// TIA Portal project "MOVIKIT_VELOCITY_V2.1_e_V15.1_V18" (V18)

(* hardware
DEVICE "S71500/ET200MP-Station_1"  S7-1500 station
   slot 0: "Profilschiene_0"  6ES7 590-1***0-0AA0
   slot 1: "S715xx"  CPU 1516F-3 PN/DP  6ES7 516-3FN00-0AB0  V1.8
DEVICE "SIMATIC 1200-Station_2"  S71200.Device
   slot 0: "S7-1200 Baugruppenträger"  Rack  V1.0
   slot 1: "S712xx"  CPU 1211C AC/DC/Rly  6ES7 211-1BD30-0XB0  V2.0
   slot 101: "CM 1243-5"  CM 1243-5  6GK7 243-5DX30-0XE0  V1.0
DEVICE "SIMATIC 300(1)"  S7-300 station
   slot 0: "Rack 0"  Rail  6ES7 390-1***0-0AA0
   slot 2: "CPU 315F-2 PN/DP"  CPU 315F-2 PN/DP  6ES7 315-2FH13-0AB0  V2.6
      slot 1: "MPI/DP interface_1"  X1
      slot 2: "PROFINET interface_1"  PN-IO
         slot 1: "Port_1"  Port
   slot 4: "DI 8/DO 8x24VDC/0.5A_1"  DI8/DO8 x 24VDC / 0.5A  6ES7 323-1BH01-0AA0
DEVICE "GSD-Geraet_4"  GSD.Device.PN
   slot 0: "Baugruppenträger"  Rack  V1.0
   slot 0: "velocity-s712xx"  MDX90 + CFN21 V4.0
      slot 0: "MDX90 + CFN21 V4.0"  MDX90 + CFN21 V4.0
      slot 1: "PN-IO"  PN-IO
         slot 1: "Port 1 - RJ45 (X40)"  Port 1 - RJ45 (X40)
         slot 2: "Port 2 - RJ45 (X41)"  Port 2 - RJ45 (X41)
   slot 2: "Modul I/O (05 Worte)_1"  Module I/O (05 words)
      slot 0: "Modul I/O (05 Worte)"  Module I/O (05 words)
DEVICE "GSD-Geraet_3"  GSD.Device.PN
   slot 0: "Baugruppenträger"  Rack  V1.0
   slot 0: "velocity-UDT-S715xx"  MDX90 + CFN21 V4.0
      slot 0: "MDX90 + CFN21 V4.0"  MDX90 + CFN21 V4.0
      slot 1: "PN-IO"  PN-IO
         slot 1: "Port 1 - RJ45 (X40)"  Port 1 - RJ45 (X40)
         slot 2: "Port 2 - RJ45 (X41)"  Port 2 - RJ45 (X41)
   slot 2: "Modul I/O (05 Worte)_1"  Module I/O (05 words)
      slot 0: "Modul I/O (05 Worte)"  Module I/O (05 words)
DEVICE "GSD-Geraet_2"  GSD.Device.PN
   slot 0: "Baugruppenträger"  Rack  V1.0
   slot 0: "velocity-UDT-s712xx"  MDX90 + CFN21 V4.0
      slot 0: "MDX90 + CFN21 V4.0"  MDX90 + CFN21 V4.0
      slot 1: "PN-IO"  PN-IO
         slot 1: "Port 1 - RJ45 (X40)"  Port 1 - RJ45 (X40)
         slot 2: "Port 2 - RJ45 (X41)"  Port 2 - RJ45 (X41)
   slot 2: "Modul I/O (05 Worte)_1"  Module I/O (05 words)
      slot 0: "Modul I/O (05 Worte)"  Module I/O (05 words)
   slot 3: "Modul I/O (01 Wort)_1"  Module I/O (01 word)
      slot 0: "Modul I/O (01 Wort)"  Module I/O (01 word)
   slot 4: "Modul I/O (02 Worte)_1"  Module I/O (02 words)
      slot 0: "Modul I/O (02 Worte)"  Module I/O (02 words)
   slot 5: "Modul I/O (05 Worte)_2"  Module I/O (05 words)
      slot 0: "Modul I/O (05 Worte)"  Module I/O (05 words)
DEVICE "GSD-Geraet_5"  GSD.Device.PN
   slot 0: "Baugruppenträger"  Rack  V1.0
   slot 0: "velocity-UDT-s73xx"  MDX90 + CFN21 V4.0
      slot 0: "MDX90 + CFN21 V4.0"  MDX90 + CFN21 V4.0
      slot 1: "PN-IO"  PN-IO
         slot 1: "Port 1 - RJ45 (X40)"  Port 1 - RJ45 (X40)
         slot 2: "Port 2 - RJ45 (X41)"  Port 2 - RJ45 (X41)
   slot 2: "Modul I/O (05 Worte)_1"  Module I/O (05 words)
      slot 0: "Modul I/O (05 Worte)"  Module I/O (05 words)
*)

// ===== PLC "S715xx"  CPU 1516F-3 PN/DP =====

VAR_GLOBAL   // PLC tag table "Standard-Variablentabelle"
   "Clock_Byte" AT %MB0 : Byte;
   "Clock_10Hz" AT %M0.0 : Bool;
   "Clock_5Hz" AT %M0.1 : Bool;
   "Clock_2.5Hz" AT %M0.2 : Bool;
   "Clock_2Hz" AT %M0.3 : Bool;
   "Clock_1.25Hz" AT %M0.4 : Bool;
   "Clock_1Hz" AT %M0.5 : Bool;
   "Clock_0.625Hz" AT %M0.6 : Bool;
   "Clock_0.5Hz" AT %M0.7 : Bool;
   "Reset" AT %M1000.0 : Bool;
   "set_ENABLE" AT %M1000.2 : Bool;
   "DRIVES_OFF" AT %M1000.1 : Bool;
   "VELOCITY_S715xx_Q" AT %A400.0 : "SEW_MOVIKIT_VelocityDrive_SETPOINTS_V2.1";   // Dieses UDT bildet die 5 Prozeßausgangsdaten der Funktion "Parameterkanal über Prozeßdaten" ab. This UDT maps the 5 process output data of the function "parameter channel via process data".
   "VELOCITY_S715xx_I" AT %E400.0 : "SEW_MOVIKIT_VelocityDrive_STATUS_V2.1";   // Dieses UDT bildet die 5 Prozeßeingangsdaten der Funktion "Parameterkanal über Prozeßdaten" ab. This UDT maps the 5 process input data of the function "parameter channel via process data"..
   "velocity-plus-S715xx _Start" AT %M1001.7 : Bool;
   "Status (FCB)" AT %MW1004 : Int;
   "SubFault_Fault" AT %MW1024 : Word;
   "Fault" AT %MB1024 : SInt;
   "SubFault" AT %MB1025 : SInt;
   "velocity-UDT-S715xx_PO1" AT %AW400 : Word;   // control word
   "velocity-UDT-S715xx_PO2" AT %QW402 : Int;   // setpoint speed
   "velocity-UDT-S715xx_PO3" AT %QW404 : Int;   // acceleration
   "velocity-UDT-S715xx_PO4" AT %QW406 : Int;   // deceleration
   "velocity-UDT-S715xx_PO5" AT %QW408 : Word;   // dig. Outputs
   "velocity-UDT-S715xx_PI1" AT %IW400 : Int;   // status word
   "velocity-UDT-S715xx_PI2" AT %IW402 : Int;   // actual speed
   "velocity-UDT-S715xx_PI3" AT %IW404 : Word;   // Status/Main/Subfault
   "velocity-UDT-S715xx_PI4" AT %IW406 : Int;   // actual torque
   "velocity-UDT-S715xx_PI5" AT %IW408 : Word;   // dig. Inputs
END_VAR

TYPE "SEW_MOVIKIT_VelocityDrive_STATUS_V2.1"
// Dieses UDT bildet die 5 Prozeßausgangsdaten des MOVIKIT VelocityDrives ab. This UDT maps the 5 process output data of the MOVIKIT VelocityDrive.
   STRUCT
      x_Bit_8_Fault : Bool;
      x_Bit_9_Warning : Bool;
      x_Bit_10_DriveTrain2_active : Bool;
      x_Bit_11_Setp_actual_speed_comp_signal_active : Bool;
      x_Bit_12_SW_Limit_switches_inactive : Bool;
      x_Bit_13_Reserved : Bool;
      x_Bit_14_StandBy_Mode_active : Bool;
      x_Bit_15_Heartbeat_OUT : Bool;
      x_Bit_0_Ready : Bool;
      x_Bit_1_STO_inactive : Bool;
      x_Bit_2_Output_Stage_enabled : Bool;
      x_Bit_3_Brake_released : Bool;
      x_Bit_4_Motor_turning : Bool;
      x_Bit_5_Active_Drive_referenced : Bool;
      x_Bit_6_New_Relative_Position_applied : Bool;
      x_Bit_7_In_Position : Bool;
      iActual_Speed : Int;
      wStatus_main_fault_sub_fault : Word;
      iActual_Torque : Int;
      wDigital_Inputs : Word;
   END_STRUCT;
END_TYPE

TYPE "SEW_MOVIKIT_VelocityDrive_SETPOINTS_V2.1"
TITLE = SEW_MOVIKIT_VelocityDrive_SETPOINTS
// Dieses UDT bildet die 5 Prozeßeingangsdaten des MOVIKIT VelocityDrives ab. This UDT maps the 5 process input data of the MOVIKIT VelocityDrive.
   STRUCT
      x_Bit_8_Fault_Reset : Bool;
      x_Bit_9_Reserved : Bool;
      x_Bit_10_Activate_DriveTrain2 : Bool;
      x_Bit_11_Reserved : Bool;
      x_Bit_12_Deactivate_SW_Limit_switches : Bool;
      x_Bit_13_Activate_Output_Stage_Inhibit : Bool;
      x_Bit_14_Activate_StandBy : Bool;
      x_Bit_15_Heartbeat_IN : Bool;
      x_Bit_0_Enable_Emergency_Stop : Bool;
      x_Bit_1_Enable_Application_Stop : Bool;
      x_Bit_2_Reserved : Bool;
      x_Bit_3_Release_Brake : Bool;
      x_Bit_4_Jog_positive : Bool;
      x_Bit_5_Jog_negative : Bool;
      x_Bit_6_Apply_relative_Position : Bool;
      x_Bit_7_Start_Stop : Bool;
      iSetpoint_Speed : Int;
      iAcceleration : Int;
      iDeceleration : Int;
      wDigital_Outputs : Word;
   END_STRUCT;
END_TYPE

FUNCTION "UDT_Velocity_Drive_example" : Void   // FC98, FBD
TITLE = Call the drive "velocity-UDT-S715xx"
{ S7_Optimized_Access := 'TRUE' }
AUTHOR : CSCEASDI
FAMILY : MOVIKIT
VERSION : 2.1
// This sample program only demonstrates the basic approach. We do not accept any legal or other liability for incorrect program functions and their consequences!
// 
// Please take note of the manual "MOVIKIT® Positioning, Velocity"
// 
// The UDTs "SEW_MOVIKIT_VelocityDrive_SETPOINTS_V2.1" and "SEW_MOVIKIT_VelocityDrive_STATUS_V2.1" are needed. Please make sure that the PLC data types are available in your TIA project. These UDTs can be copied from the original TIA sample project or from the MOVIKIT_VELOCITY_UDTs_V2.x.al14 library.
// 
// The plc tag "VELOCITY_S715xx_Q" has been assigned to the data type "SEW_MOVIKIT_VelocityDrive_SETPOINTS_V2.1" and  address Q400.0
// 
// The plc tag "VELOCITY_S715xx_I" has been assigned to the data type "SEW_MOVIKIT_VelocityDrive_STATUS_V2.1" and  address I400.0
BEGIN

REGION Network 1: Mapping of Status/Main fault/Subfault
   // If there is no fault or warning, the current FCB is output in "Status (FCB) MW1004 ).
   // 
   // If there is a fault or warning, the Subfault is copied in MB1024 and the Main fault in MB1025
   // 
   // => See "watch table "velocity-UDTSt15xx"
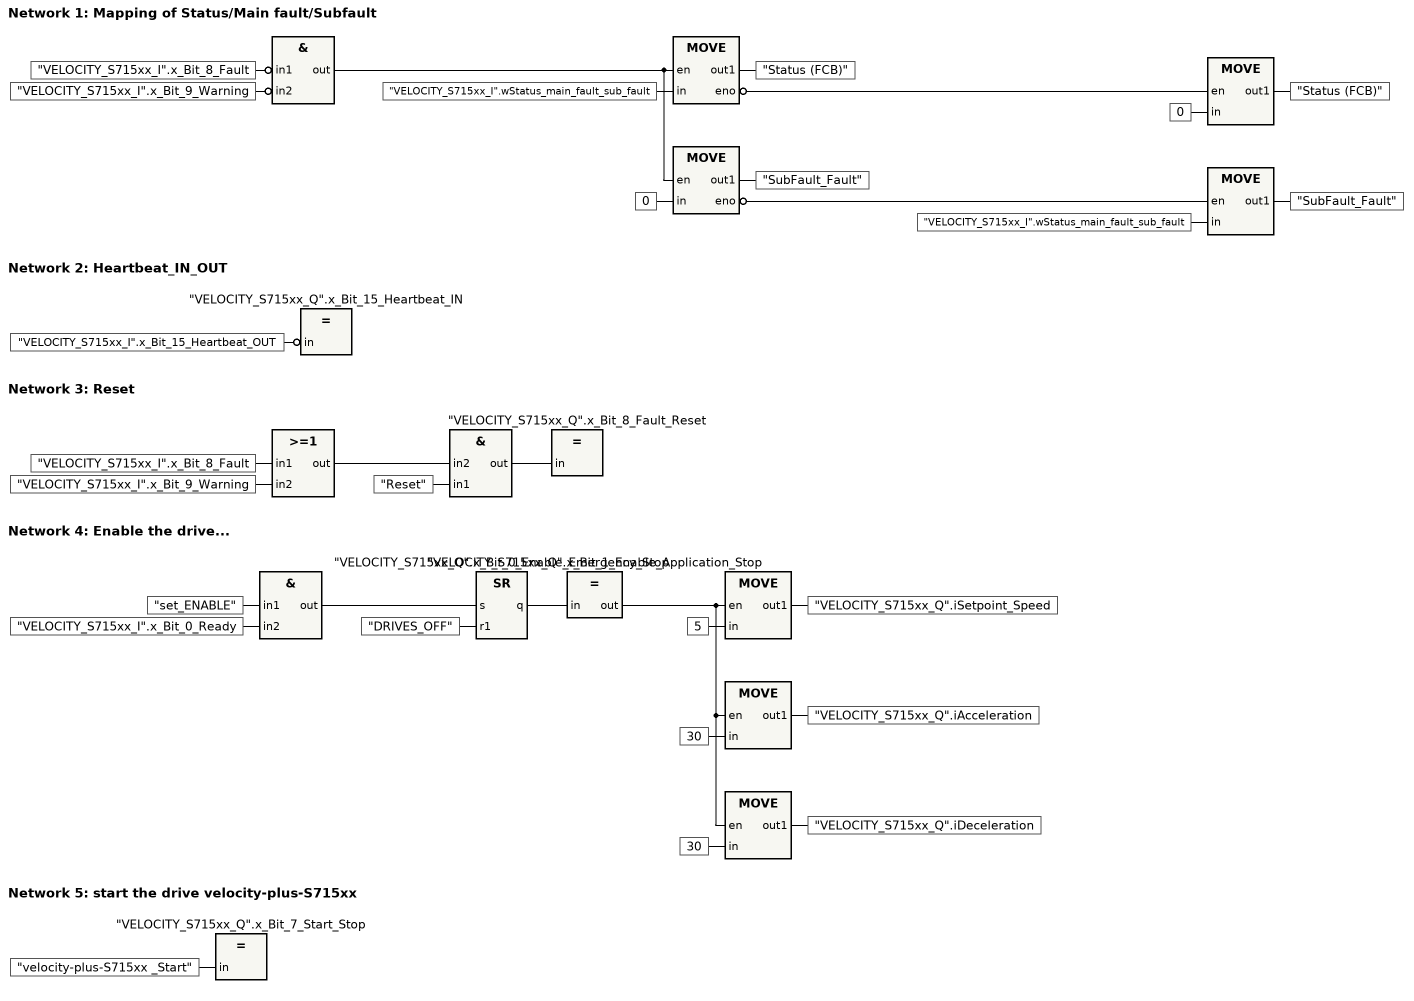
   IF NOT "VELOCITY_S715xx_I".x_Bit_8_Fault AND NOT "VELOCITY_S715xx_I".x_Bit_9_Warning THEN
       "Status (FCB)" := "VELOCITY_S715xx_I".wStatus_main_fault_sub_fault;
   END_IF;
   IF NOT (NOT "VELOCITY_S715xx_I".x_Bit_8_Fault AND NOT "VELOCITY_S715xx_I".x_Bit_9_Warning) THEN
       "Status (FCB)" := 0;
   END_IF;
   IF NOT "VELOCITY_S715xx_I".x_Bit_8_Fault AND NOT "VELOCITY_S715xx_I".x_Bit_9_Warning THEN
       "SubFault_Fault" := 0;
   END_IF;
   IF NOT (NOT "VELOCITY_S715xx_I".x_Bit_8_Fault AND NOT "VELOCITY_S715xx_I".x_Bit_9_Warning) THEN
       "SubFault_Fault" := "VELOCITY_S715xx_I".wStatus_main_fault_sub_fault;
   END_IF;
END_REGION

REGION Network 2: Heartbeat_IN_OUT
   "VELOCITY_S715xx_Q".x_Bit_15_Heartbeat_IN := NOT "VELOCITY_S715xx_I".x_Bit_15_Heartbeat_OUT;
END_REGION

REGION Network 3: Reset
   "VELOCITY_S715xx_Q".x_Bit_8_Fault_Reset := ("VELOCITY_S715xx_I".x_Bit_8_Fault OR "VELOCITY_S715xx_I".x_Bit_9_Warning) AND "Reset";
END_REGION

REGION Network 4: Enable the drive...
   // - set enable
   // - assign setpoint speed, acceleration,..,.....
   IF "set_ENABLE" AND "VELOCITY_S715xx_I".x_Bit_0_Ready THEN
       "VELOCITY_S715xx_Q".x_Bit_0_Enable_Emergency_Stop := TRUE;   // SR flip-flop
   END_IF;
   IF "DRIVES_OFF" THEN "VELOCITY_S715xx_Q".x_Bit_0_Enable_Emergency_Stop := FALSE; END_IF;
   "VELOCITY_S715xx_Q".x_Bit_1_Enable_Application_Stop := "VELOCITY_S715xx_Q".x_Bit_0_Enable_Emergency_Stop;
   IF "VELOCITY_S715xx_Q".x_Bit_0_Enable_Emergency_Stop THEN
       "VELOCITY_S715xx_Q".iSetpoint_Speed := 5;
       "VELOCITY_S715xx_Q".iAcceleration := 30;
       "VELOCITY_S715xx_Q".iDeceleration := 30;
   END_IF;
END_REGION

REGION Network 5: start the drive velocity-plus-S715xx
   "VELOCITY_S715xx_Q".x_Bit_7_Start_Stop := "velocity-plus-S715xx _Start";
END_REGION
END_FUNCTION

ORGANIZATION_BLOCK "Main"   // OB1, STL, ProgramCycle
TITLE = "Main Program Sweep (Cycle)"
{ S7_Optimized_Access := 'FALSE' }
VERSION : 0.1
// This sample program only demonstrates the basic approach. We do not accept any legal or other liability for incorrect program functions and their consequences!
// 
// Please take note of the manual "MOVIKIT® Positioning, Velocity"
   VAR_TEMP
      OB1_EV_CLASS : Byte;   // Bits 0-3 = 1 (Coming event), Bits 4-7 = 1 (Event class 1)
      OB1_SCAN_1 : Byte;   // 1 (Cold restart scan 1 of OB 1), 3 (Scan 2-n of OB 1)
      OB1_PRIORITY : Byte;   // Priority of OB Execution
      OB1_OB_NUMBR : Byte;   // 1 (Organization block 1, OB1)
      OB1_RESERVED_1 : Byte;   // Reserved for system
      OB1_RESERVED_2 : Byte;   // Reserved for system
      OB1_PREV_CYCLE : Int;   // Cycle time of previous OB1 scan (milliseconds)
      OB1_MIN_CYCLE : Int;   // Minimum cycle time of OB1 (milliseconds)
      OB1_MAX_CYCLE : Int;   // Maximum cycle time of OB1 (milliseconds)
      OB1_DATE_TIME : Date_And_Time;   // Date and time OB1 started
   END_VAR
BEGIN

REGION Network 1: Call the drive "velocity-UDT-S715xx"

         CALL  "UDT_Velocity_Drive_example";
END_REGION
END_ORGANIZATION_BLOCK

// ===== PLC "S712xx"  CPU 1211C AC/DC/Rly =====

VAR_GLOBAL   // PLC tag table "Standard-Variablentabelle"
   "Clock_Byte" AT %MB0 : Byte;
   "Clock_10Hz" AT %M0.0 : Bool;
   "Clock_5Hz" AT %M0.1 : Bool;
   "Clock_2.5Hz" AT %M0.2 : Bool;
   "Clock_2Hz" AT %M0.3 : Bool;
   "Clock_1.25Hz" AT %M0.4 : Bool;
   "Clock_1Hz" AT %M0.5 : Bool;
   "Clock_0.625Hz" AT %M0.6 : Bool;
   "Clock_0.5Hz" AT %M0.7 : Bool;
   "velocity-UDT-S712xx_PO6_Jerk_Time" AT %AW310 : Int;   // Slot 3: jerk time
   "velocity-S712xx_PO1" AT %QW326 : Int;   // control word
   "velocity-S712xx_PO2" AT %QW328 : Int;   // setpoint speed
   "velocity-S712xx_PO3" AT %QW330 : Int;   // acceleration
   "velocity-S712xx_PO4" AT %QW332 : Int;   // deceleration
   "velocity-S712xx_PO5" AT %QW334 : Int;   // dig. Outputs
   "velocity-S712xx_PI1" AT %IW326 : Int;   // status word
   "velocity-S712xx_PI2" AT %IW328 : Int;   // actual speed
   "velocity-S712xx_PI3" AT %IW330 : Int;   // Status/Main/Subfault
   "velocity-S712xx_PI4" AT %IW332 : Int;   // actual torque
   "velocity-S712xx_PI5" AT %IW334 : Int;   // dig. Inputs
   "velocity-UDT-S712xx_PO1" AT %QW300 : Int;   // Slot 2: control word
   "velocity-UDT-S712xx_PO2" AT %QW302 : Int;   // Slot 2: setpoint speed
   "velocity-UDT-S712xx_PO3" AT %QW304 : Int;   // Slot 2: acceleration
   "velocity-UDT-S712xx_PO4" AT %QW306 : Int;   // Slot 2: deceleration
   "velocity-UDT-S712xx_PO5" AT %QW308 : Int;   // Slot 2: dig. Outputs
   "velocity-UDT-S712xx_PO7" AT %QW312 : Int;   // Slot 4: control word for torque limit
   "velocity-UDT-S712xx_PO8" AT %QW314 : Int;   // Slot 4: maximum torque
   "velocity-UDT-S712xx_PO9" AT %QW316 : Int;   // Slot 5: Parameter channel control word
   "velocity-UDT-S712xx_PO10" AT %QW318 : Int;   // Slot 5: Parameter channel Index
   "velocity-UDT-S712xx_PO11" AT %QW320 : Int;   // Slot 5: Parameter channel SubIndex/Offset
   "velocity-UDT-S712xx_PO12/13" AT %QD322 : DInt;   // Slot 5: Parameter channel WriteData
   "velocity-UDT-S712xx_PI1" AT %IW300 : Int;   // Slot 2: status word
   "velocity-UDT-S712xx_PI2" AT %IW302 : Int;   // Slot 2: actual speed
   "velocity-UDT-S712xx_PI3" AT %IW304 : Int;   // Slot 2: Status/Main/Subfault
   "velocity-UDT-S712xx_PI4" AT %IW306 : Int;   // Slot 2: actual torque
   "velocity-UDT-S712xx_PI5" AT %IW308 : Int;   // Slot 2: dig. Inputs
   "velocity-UDT-S712xx_PI6" AT %IW310 : Int;   // Slot 3: res.
   "velocity-UDT-S712xx_PI7" AT %IW312 : Int;   // Slot 4: status word for torque limit
   "velocity-UDT-S712xx_PI8" AT %IW314 : Int;   // Slot 4: actual torque
   "velocity-UDT-S712xx_PI9" AT %IW316 : Int;   // Slot 5: Parameter channel status word
   "velocity-UDT-S712xx_PI10" AT %IW318 : Int;   // Slot 5: Parameter channel Index
   "velocity-UDT-S712xx_PI11" AT %IW320 : Int;   // Slot 5: Parameter channelSubIndex/Offset
   "velocity-UDT-S712xx_PI12" AT %ID322 : DInt;   // Slot 5: Parameter channel ReadData
END_VAR

TYPE "SEW_MOVIKIT_VelocityDrive_STATUS_V2.1"
// Dieses UDT bildet die 5 Prozeßausgangsdaten des MOVIKIT VelocityDrives ab. This UDT maps the 5 process output data of the MOVIKIT VelocityDrive.
   STRUCT
      x_Bit_8_Fault : Bool;
      x_Bit_9_Warning : Bool;
      x_Bit_10_DriveTrain2_active : Bool;
      x_Bit_11_Setp_actual_speed_comp_signal_active : Bool;
      x_Bit_12_SW_Limit_switches_inactive : Bool;
      x_Bit_13_Reserved : Bool;
      x_Bit_14_StandBy_Mode_active : Bool;
      x_Bit_15_Heartbeat_OUT : Bool;
      x_Bit_0_Ready : Bool;
      x_Bit_1_STO_inactive : Bool;
      x_Bit_2_Output_Stage_enabled : Bool;
      x_Bit_3_Brake_released : Bool;
      x_Bit_4_Motor_turning : Bool;
      x_Bit_5_Active_Drive_referenced : Bool;
      x_Bit_6_New_Relative_Position_applied : Bool;
      x_Bit_7_In_Position : Bool;
      iActual_Speed : Int;
      wStatus_main_fault_sub_fault : Word;
      iActual_Torque : Int;
      wDigital_Inputs : Word;
   END_STRUCT;
END_TYPE

TYPE "SEW_MOVIKIT_VelocityDrive_SETPOINTS_V2.1"
TITLE = SEW_MOVIKIT_VelocityDrive_SETPOINTS
// Dieses UDT bildet die 5 Prozeßeingangsdaten des MOVIKIT VelocityDrives ab. This UDT maps the 5 process input data of the MOVIKIT VelocityDrive.
   STRUCT
      x_Bit_8_Fault_Reset : Bool;
      x_Bit_9_Reserved : Bool;
      x_Bit_10_Activate_DriveTrain2 : Bool;
      x_Bit_11_Reserved : Bool;
      x_Bit_12_Deactivate_SW_Limit_switches : Bool;
      x_Bit_13_Activate_Output_Stage_Inhibit : Bool;
      x_Bit_14_Activate_StandBy_Mode : Bool;
      x_Bit_15_Heartbeat_IN : Bool;
      x_Bit_0_Enable_Emergency_Stop : Bool;
      x_Bit_1_Enable_Application_Stop : Bool;
      x_Bit_2_Reserved : Bool;
      x_Bit_3_Release_Brake : Bool;
      x_Bit_4_Jog_positive : Bool;
      x_Bit_5_Jog_negative : Bool;
      x_Bit_6_Apply_relative_Position : Bool;
      x_Bit_7_Start_Stop : Bool;
      iSetpoint_Speed : Int;
      iSetpoint_Acceleration : Int;
      iSetpoint_Deceleration : Int;
      wDigital_Outputs : Word;
   END_STRUCT;
END_TYPE

TYPE "SEW_MOVIKIT_5_PD_PAR_STATUS_V2.0"
   STRUCT
      x_Bit_8_READ_Service_selected : Bool;
      x_Bit_9_WRITE_Service_selected : Bool;
      x_Bit_10 : Bool;
      x_Bit_11 : Bool;
      x_Bit_12 : Bool;
      x_Bit_13_Service_active : Bool;
      x_Bit_14_Service_completed : Bool;
      x_Bit_15_Service_failed : Bool;
      x_Bit_0 : Bool;
      x_Bit_1 : Bool;
      x_Bit_2 : Bool;
      x_Bit_3 : Bool;
      x_Bit_4 : Bool;
      x_Bit_5 : Bool;
      x_Bit_6 : Bool;
      x_Bit_7 : Bool;
      i_actual_Index : Int;
      b_actual_SubIndex : Byte;
      b_actual_Offset : Byte;
      dw_value_read : DWord;
   END_STRUCT;
END_TYPE

TYPE "SEW_MOVIKIT_Function_torque_limit_STATUS_V2.0"
   STRUCT
      x_Bit_8 : Bool;
      x_Bit_9 : Bool;
      x_Bit_10 : Bool;
      x_Bit_11 : Bool;
      x_Bit_12 : Bool;
      x_Bit_13 : Bool;
      x_Bit_14 : Bool;
      x_Bit_15 : Bool;
      x_Bit_0_torque_limit_via_PD_active : Bool;
      x_Bit_1_speed_and_lag_error_monitoring_inactive : Bool;
      x_Bit_2_torque_limit_reached : Bool;
      x_Bit_3_speed_monitoring_inactive : Bool;
      x_Bit_4 : Bool;
      x_Bit_5 : Bool;
      x_Bit_6 : Bool;
      x_Bit_7 : Bool;
      i_actual_torque : Int;
   END_STRUCT;
END_TYPE

TYPE "SEW_MOVIKIT_5_PD_PAR_SETPOINTS_V2.0"
   STRUCT
      x_Bit_8_READ : Bool;
      x_Bit_9_WRITE : Bool;
      x_Bit_10 : Bool;
      x_Bit_11 : Bool;
      x_Bit_12 : Bool;
      x_Bit_13 : Bool;
      x_Bit_14_execute_function : Bool;
      x_Bit_15 : Bool;
      x_Bit_0 : Bool;
      x_Bit_1 : Bool;
      x_Bit_2 : Bool;
      x_Bit_3 : Bool;
      x_Bit_4 : Bool;
      x_Bit_5 : Bool;
      x_Bit_6 : Bool;
      x_Bit_7 : Bool;
      i_Index : Int;
      b_SubIndex : Byte;
      b_Offset : Byte;
      dw_value : DWord;
   END_STRUCT;
END_TYPE

TYPE "SEW_MOVIKIT_Function_torque_limit_SETPOINTS_V2.0"
   STRUCT
      x_Bit_8 : Bool;
      x_Bit_9 : Bool;
      x_Bit_10 : Bool;
      x_Bit_11 : Bool;
      x_Bit_12 : Bool;
      x_Bit_13 : Bool;
      x_Bit_14 : Bool;
      x_Bit_15 : Bool;
      x_Bit_0_activate_torque_limit_via_PD : Bool;
      x_Bit_1_deactivate_monitoring_of_speed_and_lag_error : Bool;
      x_Bit_2 : Bool;
      x_Bit_3_deactivate_speed_monitoring : Bool;
      x_Bit_4 : Bool;
      x_Bit_5 : Bool;
      x_Bit_6 : Bool;
      x_Bit_7 : Bool;
      i_maximum_torque : Int;
   END_STRUCT;
END_TYPE

DATA_BLOCK "Velocity_270"   // DB270
{ S7_Optimized_Access := 'FALSE' }
VERSION : 0.1
   VAR
      PO : "SEW_MOVIKIT_VelocityDrive_SETPOINTS_V2.1";
      PI : "SEW_MOVIKIT_VelocityDrive_STATUS_V2.1";
      Communication_OK : Bool;   // true: DPRD_DAT u. DPWR_DAT arbeiten fehlerfrei. false: 5-PD-Steckplatz erforderlich; Adresse an Eingang "IO_ADDRESS" überprüfen
   END_VAR
BEGIN
END_DATA_BLOCK

DATA_BLOCK "TORQUE_279"   // DB271
{ S7_Optimized_Access := 'FALSE' }
VERSION : 0.1
   VAR
      HW_IDENTIFIER : Hw_Io := 271;
      ACTIVATE_TORQUE_LIMIT_VIA_PD : Bool;
      DEACTIVATE_MONITORING_OF_SPEED_LAG_ERROR : Bool;
      DEACTIVATE_SPEED_MONITORING : Bool;
      MAXIMUM_TORQUE : Int;
      COMMUNICATION_OK : Bool;
      TORQUE_LIMIT_VIA_PD_ACTIVE : Bool;
      SPEED_LAG_ERROR_MONITORING_INACTIVE : Bool;
      TORQUE_LIMIT_REACHED : Bool;
      SPEED_MONITORING_INACTIVE : Bool;
      ACTUAL_TORQUE : Int;
   END_VAR
BEGIN
END_DATA_BLOCK

DATA_BLOCK "Velocity_290"   // DB290
{ S7_Optimized_Access := 'FALSE' }
VERSION : 0.1
   VAR
      ENABLE_RAPID_STOP : Bool;
      ENABLE_APPLICATION_STOP : Bool;
      RELEASE_BRAKE : Bool;
      START_STOP : Bool;
      RESET_ERROR : Bool;
      ACTIVATE_DRIVE_TRAIN_2 : Bool;
      DISABLE_SW_LIMIT_SWITCH : Bool;
      ACTIVATE_INHIBIT : Bool;
      ACTIVATE_STANDBY : Bool;
      SETPOINT_SPEED : Int;
      SETPOINT_ACCELERATION : Int;
      SETPOINT_DECELERATION : Int;
      DIGITAL_OUTPUTS : Word;
      COMMUNICATION_OK : Bool;
      INVERTER_READY : Bool;
      STO_INACTIVE : Bool;
      OUTPUT_STAGE_ENABLED : Bool;
      BRAKE_RELEASED : Bool;
      DRIVE_ACTIVE : Bool;
      TARGET_VALUES_ACTIVE : Bool;
      ERROR : Bool;
      WARNING : Bool;
      DRIVE_TRAIN_2_ACTIVE : Bool;
      VELOCITY_TARGET_ACTUAL_COMPARISON : Bool;
      SW_LIMIT_SWITCH_INACTIVE : Bool;
      STANDBY_ACTIVE : Bool;
      HEARTBEAT_OUT : Bool;
      ACTUAL_SPEED : Int;
      STATUS_ERROR_NO : Int;
      ACTUAL_TORQUE : Int;
      DIGITAL_INPUTS : Word;
      HEARTBEAT_IN : Bool;
   END_VAR
BEGIN
END_DATA_BLOCK

// folder: 5_PD_Parameter_channel

DATA_BLOCK "5_PD_parameter_channel_FB_DB"   // DB198
{ S7_Optimized_Access := 'FALSE' }
VERSION : 0.1
// stored: InstanceOfName 5_PD_parameter_channel_FB
"5_PD_parameter_channel_FB"
BEGIN
END_DATA_BLOCK

DATA_BLOCK "DB_5PD_PAR_272"   // DB272
{ S7_Optimized_Access := 'FALSE' }
VERSION : 0.1
   VAR
      PO : "SEW_MOVIKIT_5_PD_PAR_SETPOINTS_V2.0";
      Service : Bool;   // 0: read; 1: write
      fActivate : Bool;
      fBusy : Bool;
      fDone : Bool;
      COMMUNICATION_NOT_OK : Bool;
      TIMEOUT : Bool;
      PI : "SEW_MOVIKIT_5_PD_PAR_STATUS_V2.0";
   END_VAR
BEGIN
END_DATA_BLOCK

// folder: (top level)

FUNCTION "Call velocity-S712xx" : Void   // FC100, FBD
TITLE = Call velocity-S712xx
{ S7_Optimized_Access := 'TRUE' }
VERSION : 2.1
// This sample program only demonstrates the basic approach. We do not accept any legal or other liability for incorrect program functions and their consequences!
// 
// Please take note of the manual "MOVIKIT® Positioning, Velocity"
BEGIN

REGION Network 1: Call velocity-S712xx
   // The FC120 serves as a program module for controlling the MOVIKIT module "Velocity Drive" for the Generation C device series. With the help of the FC120, the converters can be controlled via PROFINET IO/PROFIBUS DP. 
   // 
   // Device & networks: To use this FC, a 5 PD slot must be configured.
   // 
   // Inputs of the FC:
   // 
   // "HW_Identifier": Assign the HW-Identifier of the 5 PD slot. 
   // 
   // "ENABLE_EMERGENCY_STOP" = true: Enable; false: emergency stop
   // "ENABLE_APPLICATION_STOP" = true: Enable; false: Application stop
   // "RELEASE_BRAKE" = true: release brake (without enable)
   // "START_STOP" = Start/stop with fieldbus ramp
   // "FAULT_RESET": true: Fault reset
   // "ACTIVATE_DRIVE_TRAIN_2" = true: Activate drive train 2
   // "ACTIVATE_OUPUT_STAGE_INHIBIT" = true: Activate output stage inhibit
   // "ACTIVATE_STANDBY_MODE" = true: Activate standby mode
   // "HEARTBEAT_IN": Copied to "HEARTBEAT_OUT"
   // "SETPOINT_SPEED": in user unit (INT) 
   // "SETPOINT_ACCELERATION":  in user unit (INT) 
   // "SETPOINT_DECELERATION":  in user unit (INT)
   // "DIGITAL_OUTPUTS": MoviSuite/Movikit../Inputs/Outputs: dig Outputs: the setting "control via fieldbus" is needed
   // 
   // Outputs of the FC:
   // 
   // If the data transmission/PROFINET is disrupted, all outputs will be deleted..
   // => "COMMUNICATION_OK = false (self-confirming)
   // "READY" = true: Ready for operation.
   // "STO_INACTIVE" = true: STO inactive.
   // "OUTPUT_STAGE_ENABLED" = true: Output stage enabled.
   // "BRAKE_RELEASED" = true: Brake released.
   // "MOTOR_TURNING" = true: Motor turning.
   // "FAULT" = true: Fault.
   // "WARNING" = true: Warning 
   // "DRIVE_TRAIN_2_ACTIVE" = true: Drive train 2 active.
   // "SETPOINT-ACTUAL_COMPARISON" 
   // "STANDBY_MODE_ACTIVE" = true: Stand-by Mode is active.
   // "HEARTBEAT_OUT" : This signal is copied internally from "HEARTBEAT_IN"
   // "ACTUAL_SPEED": in user unit (INT) 
   // "STATUS_MAIN_FAULT_SUB_FAULT:" (WORD)
   //    No fault: Display of current FCB; fault/warning:  High-Byte Fault; Low-Byte SubFault
   // "ACTUAL_TORQUE":in user unit (INT)
   // "DIGITAL_INPUTS" : The digital inputs are read out
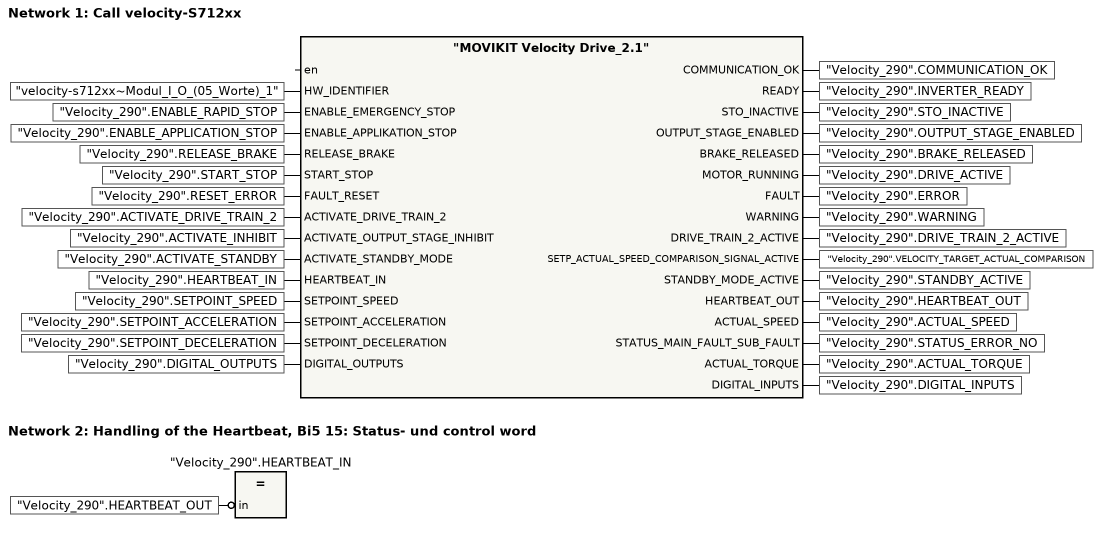
   "MOVIKIT Velocity Drive_2.1"(HW_IDENTIFIER := "velocity-s712xx~Modul_I_O_(05_Worte)_1",
                           ENABLE_EMERGENCY_STOP := "Velocity_290".ENABLE_RAPID_STOP,
                           ENABLE_APPLIKATION_STOP := "Velocity_290".ENABLE_APPLICATION_STOP,
                           RELEASE_BRAKE := "Velocity_290".RELEASE_BRAKE,
                           START_STOP := "Velocity_290".START_STOP,
                           FAULT_RESET := "Velocity_290".RESET_ERROR,
                           ACTIVATE_DRIVE_TRAIN_2 := "Velocity_290".ACTIVATE_DRIVE_TRAIN_2,
                           ACTIVATE_OUTPUT_STAGE_INHIBIT := "Velocity_290".ACTIVATE_INHIBIT,
                           ACTIVATE_STANDBY_MODE := "Velocity_290".ACTIVATE_STANDBY,
                           HEARTBEAT_IN := "Velocity_290".HEARTBEAT_IN,
                           SETPOINT_SPEED := "Velocity_290".SETPOINT_SPEED,
                           SETPOINT_ACCELERATION := "Velocity_290".SETPOINT_ACCELERATION,
                           SETPOINT_DECELERATION := "Velocity_290".SETPOINT_DECELERATION,
                           DIGITAL_OUTPUTS := "Velocity_290".DIGITAL_OUTPUTS,
                           COMMUNICATION_OK => "Velocity_290".COMMUNICATION_OK,
                           READY => "Velocity_290".INVERTER_READY,
                           STO_INACTIVE => "Velocity_290".STO_INACTIVE,
                           OUTPUT_STAGE_ENABLED => "Velocity_290".OUTPUT_STAGE_ENABLED,
                           BRAKE_RELEASED => "Velocity_290".BRAKE_RELEASED,
                           MOTOR_RUNNING => "Velocity_290".DRIVE_ACTIVE,
                           FAULT => "Velocity_290".ERROR,
                           WARNING => "Velocity_290".WARNING,
                           DRIVE_TRAIN_2_ACTIVE => "Velocity_290".DRIVE_TRAIN_2_ACTIVE,
                           SETP_ACTUAL_SPEED_COMPARISON_SIGNAL_ACTIVE => "Velocity_290".VELOCITY_TARGET_ACTUAL_COMPARISON,
                           STANDBY_MODE_ACTIVE => "Velocity_290".STANDBY_ACTIVE,
                           HEARTBEAT_OUT => "Velocity_290".HEARTBEAT_OUT,
                           ACTUAL_SPEED => "Velocity_290".ACTUAL_SPEED,
                           STATUS_MAIN_FAULT_SUB_FAULT => "Velocity_290".STATUS_ERROR_NO,
                           ACTUAL_TORQUE => "Velocity_290".ACTUAL_TORQUE,
                           DIGITAL_INPUTS => "Velocity_290".DIGITAL_INPUTS);
END_REGION

REGION Network 2: Handling of the Heartbeat, Bi5 15: Status- und control word
   "Velocity_290".HEARTBEAT_IN := NOT "Velocity_290".HEARTBEAT_OUT;
END_REGION
END_FUNCTION

FUNCTION "Call_velocity-UDT-S712xx" : Void   // FC101, FBD
TITLE = Control of the drive velocity-UDT-S712xx with the functions "Variable jerk time, Variable torque limitation.
{ S7_Optimized_Access := 'TRUE' }
VERSION : 0.1
// This sample program only demonstrates the basic approach. We do not accept any legal or other liability for incorrect program functions and their consequences!
// 
// Please take note of the manual "MOVIKIT® Positioning, Velocity"
// 
// Control of the MOVIKITS Velocity Drive with the functions "Variable jerk time and Variable torque limitation.
BEGIN

REGION Network 1: Slot 2, PD 1..5: Control of the drive velocity-UDT-S712xx
   // The FC121 serves as a program module for controlling the MOVIKIT module "Velocity Drive" for the Generation C device series. With the help of the FC121, the converters can be controlled via PROFINET IO/PROFIBUS DP. 
   // 
   // Device & networks: To use this FC, a 5 PD slot must be configured.
   // 
   // This FC uses the UDTs "SEW_MOVIKIT_VelocityDrive_SETPOINTS_V2.0" and "SEW_MOVIKIT_VelocityDrive_STATUS_V2.0". Please make sure that these PLC data types are available in your TIA project. These UDTs can be copied from the original TIA sample project or from the MOVIKIT_Vel_&_Pos_UDTs_V2.0.al14 library.
   // 
   // Inputs of the FC:
   // 
   // Attention! 
   // S71xxx: "HW_Identifier". Assign the HW-Identifier of the 5 PD slot. 
   // S73xx/4xx:"HW_Identifier"Change the data type from "HW_IO" to "WORD" Assign the peripheral address of the 5 PD slot;
   // 
   // "ENABLE_EMERGENCY_STOP" = true: Enable; false: emergency stop
   // "ENABLE_APPLICATION_STOP" = true: Enable; false: Application stop
   // "RELEASE_BRAKE" = true: release brake (without enable)
   // "START_STOP" = Start/stop with fieldbus ramp
   // "FAULT_RESET": true: Fault reset
   // "ACTIVATE_DRIVE_TRAIN_2" = true: Activate drive train 2
   // "ACTIVATE_OUPUT_STAGE_INHIBIT" = true: Activate output stage inhibit
   // "ACTIVATE_STANDBY_MODE" = true: Activate standby mode
   // "HEARTBEAT_IN": Copied to "HEARTBEAT_OUT"
   // "SETPOINT_SPEED": in user unit (INT) 
   // "SETPOINT_ACCELERATION":  in user unit (INT) 
   // "SETPOINT_DECELERATION":  in user unit (INT)
   // "DIGITAL_OUTPUTS": MoviSuite/Movikit../Inputs/Outputs: dig Outputs: the setting "control via fieldbus" is needed
   // 
   // Outputs of the FC:
   // 
   // If the data transmission/PROFINET is disrupted, all outputs will be deleted..
   // => "COMMUNICATION_OK = false (self-confirming)
   // "READY" = true: Ready for operation.
   // "STO_INACTIVE" = true: STO inactive.
   // "OUTPUT_STAGE_ENABLED" = true: Output stage enabled.
   // "BRAKE_RELEASED" = true: Brake released.
   // "MOTOR_TURNING" = true: Motor turning.
   // "FAULT" = true: Fault.
   // "WARNING" = true: Warning 
   // "DRIVE_TRAIN_2_ACTIVE" = true: Drive train 2 active.
   // "SETPOINT-ACTUAL_COMPARISON" 
   // "STANDBY_MODE_ACTIVE" = true: Stand-by Mode is active.
   // "HEARTBEAT_OUT" : This signal is copied internally from "HEARTBEAT_IN"
   // "ACTUAL_SPEED": in user unit (INT) 
   // "STATUS_MAIN_FAULT_SUB_FAULT:" (WORD)
   //    No fault: Display of current FCB; fault/warning:  High-Byte Fault; Low-Byte SubFault
   // "ACTUAL_TORQUE":in user unit (INT)
   // "DIGITAL_INPUTS" : The digital inputs are read out
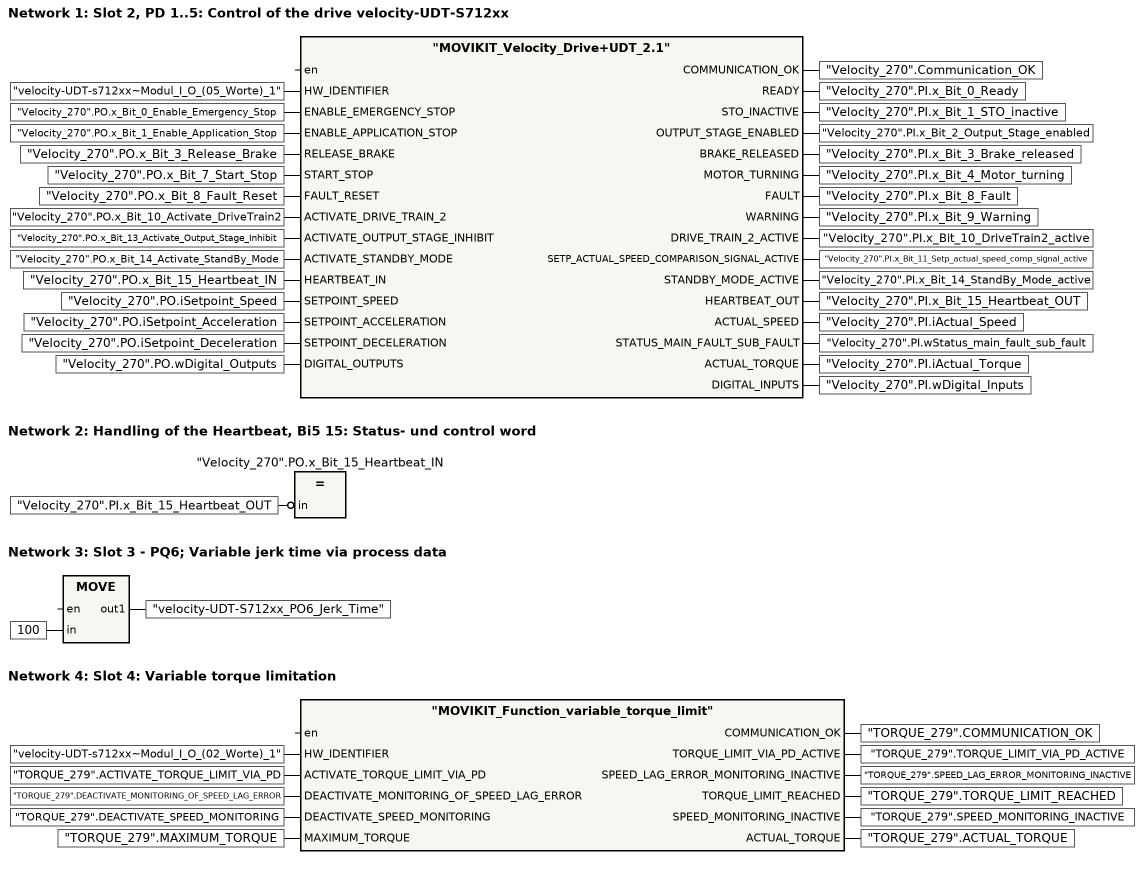
   "MOVIKIT_Velocity_Drive+UDT_2.1"(HW_IDENTIFIER := "velocity-UDT-s712xx~Modul_I_O_(05_Worte)_1",
                           ENABLE_EMERGENCY_STOP := "Velocity_270".PO.x_Bit_0_Enable_Emergency_Stop,
                           ENABLE_APPLICATION_STOP := "Velocity_270".PO.x_Bit_1_Enable_Application_Stop,
                           RELEASE_BRAKE := "Velocity_270".PO.x_Bit_3_Release_Brake,
                           START_STOP := "Velocity_270".PO.x_Bit_7_Start_Stop,
                           FAULT_RESET := "Velocity_270".PO.x_Bit_8_Fault_Reset,
                           ACTIVATE_DRIVE_TRAIN_2 := "Velocity_270".PO.x_Bit_10_Activate_DriveTrain2,
                           ACTIVATE_OUTPUT_STAGE_INHIBIT := "Velocity_270".PO.x_Bit_13_Activate_Output_Stage_Inhibit,
                           ACTIVATE_STANDBY_MODE := "Velocity_270".PO.x_Bit_14_Activate_StandBy_Mode,
                           HEARTBEAT_IN := "Velocity_270".PO.x_Bit_15_Heartbeat_IN,
                           SETPOINT_SPEED := "Velocity_270".PO.iSetpoint_Speed,
                           SETPOINT_ACCELERATION := "Velocity_270".PO.iSetpoint_Acceleration,
                           SETPOINT_DECELERATION := "Velocity_270".PO.iSetpoint_Deceleration,
                           DIGITAL_OUTPUTS := "Velocity_270".PO.wDigital_Outputs,
                           COMMUNICATION_OK => "Velocity_270".Communication_OK,
                           READY => "Velocity_270".PI.x_Bit_0_Ready,
                           STO_INACTIVE => "Velocity_270".PI.x_Bit_1_STO_inactive,
                           OUTPUT_STAGE_ENABLED => "Velocity_270".PI.x_Bit_2_Output_Stage_enabled,
                           BRAKE_RELEASED => "Velocity_270".PI.x_Bit_3_Brake_released,
                           MOTOR_TURNING => "Velocity_270".PI.x_Bit_4_Motor_turning,
                           FAULT => "Velocity_270".PI.x_Bit_8_Fault,
                           WARNING => "Velocity_270".PI.x_Bit_9_Warning,
                           DRIVE_TRAIN_2_ACTIVE => "Velocity_270".PI.x_Bit_10_DriveTrain2_active,
                           SETP_ACTUAL_SPEED_COMPARISON_SIGNAL_ACTIVE => "Velocity_270".PI.x_Bit_11_Setp_actual_speed_comp_signal_active,
                           STANDBY_MODE_ACTIVE => "Velocity_270".PI.x_Bit_14_StandBy_Mode_active,
                           HEARTBEAT_OUT => "Velocity_270".PI.x_Bit_15_Heartbeat_OUT,
                           ACTUAL_SPEED => "Velocity_270".PI.iActual_Speed,
                           STATUS_MAIN_FAULT_SUB_FAULT => "Velocity_270".PI.wStatus_main_fault_sub_fault,
                           ACTUAL_TORQUE => "Velocity_270".PI.iActual_Torque,
                           DIGITAL_INPUTS => "Velocity_270".PI.wDigital_Inputs);
END_REGION

REGION Network 2: Handling of the Heartbeat, Bi5 15: Status- und control word
   "Velocity_270".PO.x_Bit_15_Heartbeat_IN := NOT "Velocity_270".PI.x_Bit_15_Heartbeat_OUT;
END_REGION

REGION Network 3: Slot 3 - PQ6; Variable jerk time via process data
   // This additional function extends the range of functions
   // by providing the ability to specify the jerk time.
   // The additional function extends the process data
   // length by one process data word.
   // 
   // The jerk is written directly on the output word:
   "velocity-UDT-S712xx_PO6_Jerk_Time" := 100;
END_REGION

REGION Network 4: Slot 4: Variable torque limitation
   // The additional function "Variable torque limiting Q1" lets you specify the torque via the
   // application in 0.1% × nominal motor torque. For fieldbus
   // operation, the process data length is extended by 2 process data words.
   // 
   // This FC uses the UDTs "SEW_Movikit_Function_torque_limit_SETPOINTS_V2.0" and "SEW_MOVIKIT_Function_torque_limit_STATUS_V2.0". 
   // Please make sure that these PLC data types are available in your TIA project.
   // These UDTs can be copied from the original TIA sample project or from the MOVIKIT_Vel_&_Pos_UDTs_V2.0.al14 library.
   // 
   // Inputs of the FC:
   // 
   // Attention! 
   // S71xxx: "HW_Identifier". Assign the HW-Identifier of the 2 PD slot. 
   // S73xx/4xx:"HW_Identifier"Change the data type from "HW_IO" to "WORD" Assign the peripheral address of the 2 PD slot;
   // 
   // "ACTIVATE_TORQUE_LIMIT_VIA_PD": Activation of torque limiting
   // "DEACTIVATE_MONITORING_OF_SPEED_LAG_ERROR": Deactivation of monitoring for speed and lag error
   // "DEACTIVATE_SPEED_MONITORING": Deactivation of speed monitoring
   // "MAXIMUM_TORQUE": Torque related to the nominal motor torque (unit: 0.1%)
   // 
   // Outputs of the FC:
   // 
   // If the data transmission/PROFINET is disrupted, all outputs will be deleted..
   // => "COMMUNICATION_OK = false (self-confirming)
   // "TORQUE_LIMIT_VIA_PD_ACTIVE": Torque limit via PD active
   // "SPEED_LAG_ERROR_MONITORING_INACTIVE": Speed and lag error inactive
   // "TORQUE_LIMIT_REACHED": Torque limit reached
   // "SPEED_MONITORING_INACTIVE": Speed monitoring inactive
   // "ACTUAL_TORQUE": Current torque in relation to the nominal motor torque (unit: 0.1%)
   "MOVIKIT_Function_variable_torque_limit"(HW_IDENTIFIER := "velocity-UDT-s712xx~Modul_I_O_(02_Worte)_1",
                           ACTIVATE_TORQUE_LIMIT_VIA_PD := "TORQUE_279".ACTIVATE_TORQUE_LIMIT_VIA_PD,
                           DEACTIVATE_MONITORING_OF_SPEED_LAG_ERROR := "TORQUE_279".DEACTIVATE_MONITORING_OF_SPEED_LAG_ERROR,
                           DEACTIVATE_SPEED_MONITORING := "TORQUE_279".DEACTIVATE_SPEED_MONITORING,
                           MAXIMUM_TORQUE := "TORQUE_279".MAXIMUM_TORQUE,
                           COMMUNICATION_OK => "TORQUE_279".COMMUNICATION_OK,
                           TORQUE_LIMIT_VIA_PD_ACTIVE => "TORQUE_279".TORQUE_LIMIT_VIA_PD_ACTIVE,
                           SPEED_LAG_ERROR_MONITORING_INACTIVE => "TORQUE_279".SPEED_LAG_ERROR_MONITORING_INACTIVE,
                           TORQUE_LIMIT_REACHED => "TORQUE_279".TORQUE_LIMIT_REACHED,
                           SPEED_MONITORING_INACTIVE => "TORQUE_279".SPEED_MONITORING_INACTIVE,
                           ACTUAL_TORQUE => "TORQUE_279".ACTUAL_TORQUE);
END_REGION
END_FUNCTION

FUNCTION "MOVIKIT Velocity Drive_2.1" : Void   // FC120, SCL
TITLE = MOVIKIT Velocity Drive_2.1
{ S7_Optimized_Access := 'TRUE' }
AUTHOR : SVSPASE
FAMILY : MOVIKIT
VERSION : 2.1
// This sample program only demonstrates the basic approach. We do not accept any legal or other liability for incorrect program functions and their consequences!
// 
// The FC120 serves as a program module for controlling the MOVIKIT module "Velocity Drive" for the Generation C device series. With the help of the FC120,
// the converters can be controlled via PROFINET IO/PROFIBUS DP.
// 
// Device & networks: To use this FC, a 5 PD slot must be configured.
// 
// Attention Input "HW_Identifier":
// Assign the HW-Identifier of the 5 PD slot.
   VAR_INPUT
      HW_IDENTIFIER : Hw_Io;   // S71xxx: Assign the HW-Identifier of the 5 PD slot.
      ENABLE_EMERGENCY_STOP : Bool;   // true: Enable; false: emergency stop
      ENABLE_APPLIKATION_STOP : Bool;   // true: Enable; false: Application stop
      RELEASE_BRAKE : Bool;   // true: release brake (without enable)
      START_STOP : Bool;   // Start/stop with fieldbus ramp
      FAULT_RESET : Bool;   // true: Fault reset
      ACTIVATE_DRIVE_TRAIN_2 : Bool;   // true: Activate drive train 2
      ACTIVATE_OUTPUT_STAGE_INHIBIT : Bool;   // true: Activate output stage inhibit
      ACTIVATE_STANDBY_MODE : Bool;   // true: Activate standby mode
      HEARTBEAT_IN : Bool;   // Copied to HEARTBEAT_OUT
      SETPOINT_SPEED : Int;   // in user unit (INT)
      SETPOINT_ACCELERATION : Int;   // in user unit (INT)
      SETPOINT_DECELERATION : Int;   // in user unit (INT)
      DIGITAL_OUTPUTS : Word;   // MoviSuite/Movikit../Inputs/Outputs: dig Outputs: the setting "control via fieldbus" is needed
   END_VAR
   VAR_OUTPUT
      COMMUNICATION_OK : Bool;   // true: DPRD_DAT and DPWR_DAT are working correctly. false: 5 PD slot required; Check input "HW_Identifier
      READY : Bool;   // true: Ready for operation.
      STO_INACTIVE : Bool;   // true: STO inactive.
      OUTPUT_STAGE_ENABLED : Bool;   // true: Output stage enabled.
      BRAKE_RELEASED : Bool;   // true: Brake released.
      MOTOR_RUNNING : Bool;   // true: Motor running.
      FAULT : Bool;   // true: Fault.
      WARNING : Bool;   // true: Warning
      DRIVE_TRAIN_2_ACTIVE : Bool;   // true: Drive train 2 active.
      SETP_ACTUAL_SPEED_COMPARISON_SIGNAL_ACTIVE : Bool;
      STANDBY_MODE_ACTIVE : Bool;   // true: Stand-by Mode is active.
      HEARTBEAT_OUT : Bool;   // This signal is copied internally from "HEARTBEAT_IN"
      ACTUAL_SPEED : Int;   // in user unit (INT)
      STATUS_MAIN_FAULT_SUB_FAULT : Word;   // No fault: Display of current FCB; fault/warning: High-Byte Fault; Low-Byte SubFault
      ACTUAL_TORQUE : Int;   // in user unit (INT)
      DIGITAL_INPUTS : Word;   // The binary inputs are read out
   END_VAR
   VAR_TEMP
      PI : Array[1..5] of Word;
      PO : Array[1..5] of Word;
      DPRD_RET_VAL : Int;
      DPWR_RET_VAL : Int;
   END_VAR
BEGIN
   (*This sample program only demonstrates the basic approach. We do not accept any legal or other liability for incorrect program functions and their consequences!

   The FC120 serves as a program module for controlling the MOVIKIT module "Velocity Drive" for the Generation C device series. With the help of the FC120,
   the converters can be controlled via PROFINET IO/PROFIBUS DP.

   Device & networks: To use this FC, a 5 PD slot must be configured.

   Attention Input "HW_Identifier":
   Assign the HW-Identifier of the 5 PD slot. 
   *)

   //DPRD_DAT: Reading Consistent Data of a DP Standard Slave/PROFINET IO device
   #DPRD_RET_VAL:=DPRD_DAT(LADDR:=#HW_IDENTIFIER, RECORD=>#PI);


   IF #DPRD_RET_VAL = 0 THEN //If no error occurs while the instruction is being executed...

       #COMMUNICATION_OK := TRUE;

       //Mapping the signals of the Status word:
       #READY := #PI[1].%X0;
       #STO_INACTIVE := #PI[1].%X1;
       #OUTPUT_STAGE_ENABLED := #PI[1].%X2;
       #BRAKE_RELEASED := #PI[1].%X3;
       #MOTOR_RUNNING := #PI[1].%X4;
       #FAULT := #PI[1].%X8;
       #WARNING := #PI[1].%X9;
       #DRIVE_TRAIN_2_ACTIVE := #PI[1].%X10;
       #SETP_ACTUAL_SPEED_COMPARISON_SIGNAL_ACTIVE := #PI[1].%X11;
       #STANDBY_MODE_ACTIVE := #PI[1].%X14;
       #HEARTBEAT_OUT := #PI[1].%X15;

       //Assign PI2..5
       #ACTUAL_SPEED := WORD_TO_INT(#PI[2]);
       #STATUS_MAIN_FAULT_SUB_FAULT := #PI[3];
       #ACTUAL_TORQUE := WORD_TO_INT(#PI[4]) ;
       #DIGITAL_INPUTS := #PI[5];

       //Mapping the signals of the control word:
       #PO[1].%X0 := #ENABLE_EMERGENCY_STOP;
       #PO[1].%X1 := #ENABLE_APPLIKATION_STOP;
       #PO[1].%X3 := #RELEASE_BRAKE;
       #PO[1].%X7 := #START_STOP;
       #PO[1].%X8 := #FAULT_RESET;
       #PO[1].%X10 := #ACTIVATE_DRIVE_TRAIN_2;
       #PO[1].%X13 := #ACTIVATE_OUTPUT_STAGE_INHIBIT;
       #PO[1].%X14 := #ACTIVATE_STANDBY_MODE;
       #PO[1].%X15 := #HEARTBEAT_IN;

       //Set the not used Bits to "false"
       #PO[1].%X2 := FALSE;
       #PO[1].%X4 := FALSE;
       #PO[1].%X5 := FALSE;
       #PO[1].%X6 := FALSE;
       #PO[1].%X9 := FALSE;
       #PO[1].%X11 := FALSE;
       #PO[1].%X12 := FALSE;

       //Assig the POs 2..5
       #PO[2] := INT_TO_WORD(#SETPOINT_SPEED);
       #PO[3] := INT_TO_WORD(#SETPOINT_ACCELERATION);
       #PO[4] := INT_TO_WORD(#SETPOINT_DECELERATION);
       #PO[5] := #DIGITAL_OUTPUTS;

   ELSE
       GOTO END;
   END_IF;

   //DPWR_DAT: Write consistent data of a DP standard slave/PROFINET IO device
   #DPWR_RET_VAL := DPWR_DAT(LADDR := #HW_IDENTIFIER, RECORD := #PO);

   END:
   IF #DPRD_RET_VAL <> 0 OR #DPWR_RET_VAL <> 0 THEN
       #COMMUNICATION_OK := FALSE;
       //Erase FC outputs in case of an error
       #READY := FALSE;
       #STO_INACTIVE := FALSE;
       #OUTPUT_STAGE_ENABLED := FALSE;
       #BRAKE_RELEASED := FALSE;
       #MOTOR_RUNNING := FALSE;
       #FAULT := FALSE;
       #WARNING := FALSE;
       #DRIVE_TRAIN_2_ACTIVE := FALSE;
       #SETP_ACTUAL_SPEED_COMPARISON_SIGNAL_ACTIVE := FALSE;
       #STANDBY_MODE_ACTIVE := FALSE;
       #HEARTBEAT_OUT := FALSE;
       #ACTUAL_SPEED := 0;
       #STATUS_MAIN_FAULT_SUB_FAULT := 0;
       #ACTUAL_TORQUE := 0;
       #DIGITAL_INPUTS := 0;
   END_IF;
END_FUNCTION

FUNCTION "MOVIKIT_Velocity_Drive+UDT_2.1" : Void   // FC121, SCL
TITLE = Movikit_Velocity_Drive+UDT_2.1
{ S7_Optimized_Access := 'FALSE' }
AUTHOR : SVSPASE
FAMILY : MOVIKIT
VERSION : 2.1
// This sample program only demonstrates the basic approach. We do not accept any legal or other liability for incorrect program functions and their consequences!
// 
// The FC121 serves as a program module for controlling the MOVIKIT module "Velocity Drive+UDT" for the Generation C device series. With the help of the FC121,
// the converters can be controlled via PROFINET IO/PROFIBUS DP.
// 
// Device & networks: To use this FC, a 5 PD slot must be configured.
// 
// This FC uses the UDTs SEW_MOVIKIT_VelocityDrive_SETPOINTS_V2.1 and SEW_MOVIKIT_VelocityDrive_STATUS_V2.1. 
// Please make sure that these PLC data types are available in your TIA project.
// These UDTs can be copied from the original TIA sample project or from the MOVIKIT_Vel_&_Pos_UDTs_V2.x.al14 library.
// 
// Attention Input "HW_Identifier":
// Assign the HW-Identifier of the 5 PD slot. S73xx/4xx:Change Data type from HW_IO to WORD;  Assign the peripheral address of the 5 PD slot
   VAR_INPUT
      HW_IDENTIFIER : Hw_Io;   // S71xxx: Assign the HW-Identifier of the 5 PD slot. S73xx/4xx:Change Data type from HW_IO to WORD; Assign the peripheral address of the 5 PD slot
      ENABLE_EMERGENCY_STOP : Bool;   // true: Enable; false: emergency stop
      ENABLE_APPLICATION_STOP : Bool;   // true: Enable; false: Application stop
      RELEASE_BRAKE : Bool;   // true: release brake (without enable)
      START_STOP : Bool;   // Start/stop with fieldbus ramp
      FAULT_RESET : Bool;   // true: Fault reset
      ACTIVATE_DRIVE_TRAIN_2 : Bool;   // true: Activate drive train 2
      ACTIVATE_OUTPUT_STAGE_INHIBIT : Bool;   // true: Activate output stage inhibit
      ACTIVATE_STANDBY_MODE : Bool;   // true: Activate standby mode
      HEARTBEAT_IN : Bool;   // Copied to "HEARTBEAT_OUT"
      SETPOINT_SPEED : Int;   // in user unit (INT)
      SETPOINT_ACCELERATION : Int;   // in user unit (INT)
      SETPOINT_DECELERATION : Int;   // in user unit (INT)
      DIGITAL_OUTPUTS : Word;   // MoviSuite/Movikit../Inputs/Outputs: dig Outputs: the setting "control via fieldbus" is needed
   END_VAR
   VAR_OUTPUT
      COMMUNICATION_OK : Bool;   // true: DPRD_DAT and DPWR_DAT are working correctly. false: 5 PD slot required; Check input "HW_Identifier"
      READY : Bool;   // true: Ready for operation.
      STO_INACTIVE : Bool;   // true: STO inactive.
      OUTPUT_STAGE_ENABLED : Bool;   // true: Output stage enabled.
      BRAKE_RELEASED : Bool;   // true: Brake released.
      MOTOR_TURNING : Bool;   // true: Motor running.
      FAULT : Bool;   // true: Fault.
      WARNING : Bool;   // true: Warning
      DRIVE_TRAIN_2_ACTIVE : Bool;   // true: Drive train 2 active.
      SETP_ACTUAL_SPEED_COMPARISON_SIGNAL_ACTIVE : Bool;
      STANDBY_MODE_ACTIVE : Bool;   // true: Stand-by Mode is active.
      HEARTBEAT_OUT : Bool;   // This signal is copied internally from "HEARTBEAT_IN"
      ACTUAL_SPEED : Int;   // in user unit (INT)
      STATUS_MAIN_FAULT_SUB_FAULT : Word;   // No fault: Display of current FCB; fault/warning: High-Byte Fault; Low-Byte SubFault
      ACTUAL_TORQUE : Int;   // in user unit (INT)
      DIGITAL_INPUTS : Word;   // The digital inputs are read out
   END_VAR
   VAR_TEMP
      PI : "SEW_MOVIKIT_VelocityDrive_STATUS_V2.1";   // Dieses UDT bildet die 5 Prozeßeingangsdaten des MOVIKIT VelocityDrives ab. This UDT maps the 5 process input data of the MOVIKIT VelocityDrive.
      PO : "SEW_MOVIKIT_VelocityDrive_SETPOINTS_V2.1";   // Dieses UDT bildet die 5 Prozeßausgangsdaten des MOVIKIT VelocityDrives ab. This UDT maps the 5 process output data of the MOVIKIT VelocityDrive.
      DPRD_RET_VAL : Int;
      DPWR_RET_VAL : Int;
   END_VAR
BEGIN
   (*This sample program only demonstrates the basic approach. We do not accept any legal or other liability for incorrect program functions and their consequences!

   The FC121 serves as a program module for controlling the MOVIKIT module "Velocity Drive+UDT" for the Generation C device series. With the help of the FC121,
   the converters can be controlled via PROFINET IO/PROFIBUS DP.

   Device & networks: To use this FC, a 5 PD slot must be configured.

   This FC uses the UDTs SEW_MOVIKIT_VelocityDrive_SETPOINTS_V2.1 and SEW_MOVIKIT_VelocityDrive_STATUS_V2.1. 
   Please make sure that these PLC data types are available in your TIA project.
   These UDTs can be copied from the original TIA sample project or from the MOVIKIT_Vel_&_Pos_UDTs_V2.x.al14 library.

   Attention Input "HW_Identifier":
   Assign the HW-Identifier of the 5 PD slot. S73xx/4xx:Change Data type from HW_IO to WORD;  Assign the peripheral address of the 5 PD slot
   *)

   //DPRD_DAT: Reading Consistent Data of a DP Standard Slave/PROFINET IO device
   #DPRD_RET_VAL := DPRD_DAT(LADDR := #HW_IDENTIFIER, RECORD => #PI);


   IF #DPRD_RET_VAL = 0 THEN //If no error occurs while the instruction is being executed...
       #COMMUNICATION_OK := TRUE;

       //Mapping the signals of the Status word:
       #READY := #PI.x_Bit_0_Ready;
       #STO_INACTIVE := #PI.x_Bit_1_STO_inactive;
       #OUTPUT_STAGE_ENABLED := #PI.x_Bit_2_Output_Stage_enabled;
       #BRAKE_RELEASED := #PI.x_Bit_3_Brake_released;
       #MOTOR_TURNING :=#PI.x_Bit_4_Motor_turning;
       #FAULT := #PI.x_Bit_8_Fault;
       #WARNING := #PI.x_Bit_9_Warning;
       #DRIVE_TRAIN_2_ACTIVE := #PI.x_Bit_10_DriveTrain2_active;
       #SETP_ACTUAL_SPEED_COMPARISON_SIGNAL_ACTIVE := #PI.x_Bit_11_Setp_actual_speed_comp_signal_active;
       #STANDBY_MODE_ACTIVE := #PI.x_Bit_14_StandBy_Mode_active;
       #HEARTBEAT_OUT := #PI.x_Bit_15_Heartbeat_OUT;

       //Assign PI2..5
       #ACTUAL_SPEED := #PI.iActual_Speed;
       #STATUS_MAIN_FAULT_SUB_FAULT := #PI.wStatus_main_fault_sub_fault;
       #ACTUAL_TORQUE := #PI.iActual_Torque;
       #DIGITAL_INPUTS := #PI.wDigital_Inputs;

       //Mapping the signals of the control word:
       #PO.x_Bit_0_Enable_Emergency_Stop:= #ENABLE_EMERGENCY_STOP;
       #PO.x_Bit_1_Enable_Application_Stop := #ENABLE_APPLICATION_STOP;
       #PO.x_Bit_3_Release_Brake:= #RELEASE_BRAKE;
       #PO.x_Bit_7_Start_Stop:= #START_STOP;
       #PO.x_Bit_8_Fault_Reset := #FAULT_RESET;
       #PO.x_Bit_10_Activate_DriveTrain2 := #ACTIVATE_DRIVE_TRAIN_2;
       #PO.x_Bit_13_Activate_Output_Stage_Inhibit := #ACTIVATE_OUTPUT_STAGE_INHIBIT;
       #PO.x_Bit_14_Activate_StandBy_Mode := #ACTIVATE_STANDBY_MODE;
       #PO.x_Bit_15_Heartbeat_IN := #HEARTBEAT_IN;

       //Set the not used Bits to "false"
       #PO.x_Bit_2_Reserved:= FALSE;
       #PO.x_Bit_4_Jog_positive := FALSE;
       #PO.x_Bit_5_Jog_negative  := FALSE;
       #PO.x_Bit_6_Apply_relative_Position := FALSE;
       #PO.x_Bit_9_Reserved := FALSE;
       #PO.x_Bit_11_Reserved := FALSE;
       #PO.x_Bit_12_Deactivate_SW_Limit_switches := false;

       //Assig the POs 2..5
       #PO.iSetpoint_Speed := #SETPOINT_SPEED;
       #PO.iSetpoint_Acceleration := #SETPOINT_ACCELERATION;
       #PO.iSetpoint_Deceleration := #SETPOINT_DECELERATION;
       #PO.wDigital_Outputs := #DIGITAL_OUTPUTS;

   ELSE
       GOTO END;
   END_IF;

   //DPWR_DAT: Write consistent data of a DP standard slave/PROFINET IO device
   #DPWR_RET_VAL := DPWR_DAT(LADDR := #HW_IDENTIFIER, RECORD := #PO);

   END:
   IF #DPRD_RET_VAL <> 0 OR #DPWR_RET_VAL <> 0 THEN
       #COMMUNICATION_OK := FALSE;
       //Erase FC outputs in case of an error
       #READY := FALSE;
       #STO_INACTIVE := FALSE;
       #OUTPUT_STAGE_ENABLED := FALSE;
       #BRAKE_RELEASED := FALSE;
       #MOTOR_TURNING := FALSE;
       #FAULT := FALSE;
       #WARNING := FALSE;
       #DRIVE_TRAIN_2_ACTIVE := FALSE;
       #SETP_ACTUAL_SPEED_COMPARISON_SIGNAL_ACTIVE := FALSE;
       #STANDBY_MODE_ACTIVE := FALSE;
       #HEARTBEAT_OUT := FALSE;
       #ACTUAL_SPEED := 0;
       #STATUS_MAIN_FAULT_SUB_FAULT := 0;
       #ACTUAL_TORQUE := 0;
       #DIGITAL_INPUTS := 0;
   END_IF;
END_FUNCTION

FUNCTION "MOVIKIT_Function_variable_torque_limit" : Void   // FC191, SCL
TITLE = Movikit_Function_variable_torque_limit
{ S7_Optimized_Access := 'FALSE' }
AUTHOR : SVSPASE
FAMILY : MOVIKIT
VERSION : 2.0
// This sample program only demonstrates the basic approach. We do not accept any legal or other liability for incorrect program functions and their consequences!
// 
// This FC is used to control the MOVIKIT function "variable torque limit Q1 (2PD)"
// 
// Device & networks: To use this FC, a 2 PD slot must be configured.
// 
// This FC uses the UDTs "SEW_Movikit_Function_torque_limit_SETPOINTS_V2.0" and "SEW_MOVIKIT_Function_torque_limit_STATUS_V2.0". 
// Please make sure that these PLC data types are available in your TIA project.
// These UDTs can be copied from the original TIA sample project or from the MOVIKIT_Vel_&_Pos_UDTs_V2.0.al14 library.
// 
// Attention Input "HW_Identifier":
// Assign the HW-Identifier of the 2 PD slot. S73xx/4xx:Change Data type from HW_IO to WORD;  Assign the peripheral address of the 2 PD slot
   VAR_INPUT
      HW_IDENTIFIER : Hw_Io;   // S71xxx: Assign the HW-Identifier of the 2 PD slot. S73xx/4xx:Change Data type from HW_IO to WORD; Assign the peripheral address of the 2 PD slot
      ACTIVATE_TORQUE_LIMIT_VIA_PD : Bool;   // activate torque limit via PD
      DEACTIVATE_MONITORING_OF_SPEED_LAG_ERROR : Bool;   // deactivate monitoring of lag and speed errors
      DEACTIVATE_SPEED_MONITORING : Bool;   // deactivate speed monitoring
      MAXIMUM_TORQUE : Int;   // maximum torque
   END_VAR
   VAR_OUTPUT
      COMMUNICATION_OK : Bool;
      TORQUE_LIMIT_VIA_PD_ACTIVE : Bool;   // Torque limit via PD active
      SPEED_LAG_ERROR_MONITORING_INACTIVE : Bool;   // Speed and lag error inactive
      TORQUE_LIMIT_REACHED : Bool;   // Torque limit reached
      SPEED_MONITORING_INACTIVE : Bool;   // Speed monitoring inactive
      ACTUAL_TORQUE : Int;   // Actual torque
   END_VAR
   VAR_TEMP
      PI : "SEW_MOVIKIT_Function_torque_limit_STATUS_V2.0";
      PO : "SEW_MOVIKIT_Function_torque_limit_SETPOINTS_V2.0";
      DPRD_RET_VAL : Int;
      DPWR_RET_VAL : Int;
   END_VAR
BEGIN
   (*This sample program only demonstrates the basic approach. We do not accept any legal or other liability for incorrect program functions and their consequences!

   This FC is used to control the MOVIKIT function "variable torque limit Q1 (2PD)"

   Device & networks: To use this FC, a 2 PD slot must be configured.

   This FC uses the UDTs "SEW_Movikit_Function_torque_limit_SETPOINTS_V2.0" and "SEW_MOVIKIT_Function_torque_limit_STATUS_V2.0". 
   Please make sure that these PLC data types are available in your TIA project.
   These UDTs can be copied from the original TIA sample project or from the MOVIKIT_Vel_&_Pos_UDTs_V2.0.al14 library.

   Attention Input "HW_Identifier":
   Assign the HW-Identifier of the 2 PD slot. S73xx/4xx:Change Data type from HW_IO to WORD;  Assign the peripheral address of the 2 PD slot*)



   //DPWR_DAT: Write consistent data of a DP standard slave/PROFINET IO device
   #DPRD_RET_VAL := DPRD_DAT(LADDR := #HW_IDENTIFIER, RECORD => #PI);


   IF #DPRD_RET_VAL = 0 THEN
       #COMMUNICATION_OK := TRUE;

       //Mapping the signals of the Status word:
       #TORQUE_LIMIT_VIA_PD_ACTIVE := #PI.x_Bit_0_torque_limit_via_PD_active;
       #SPEED_LAG_ERROR_MONITORING_INACTIVE := #PI.x_Bit_1_speed_and_lag_error_monitoring_inactive;
       #TORQUE_LIMIT_REACHED := #PI.x_Bit_2_torque_limit_reached;
       #SPEED_MONITORING_INACTIVE := #PI.x_Bit_3_speed_monitoring_inactive;

       //Zuweisen der Ausgangsworte des Bausteins
       #ACTUAL_TORQUE := #PI.i_actual_torque;

       //Mapping the signals of the control word:
       #PO.x_Bit_0_activate_torque_limit_via_PD := #ACTIVATE_TORQUE_LIMIT_VIA_PD;
       #PO.x_Bit_1_deactivate_monitoring_of_speed_and_lag_error:= #DEACTIVATE_MONITORING_OF_SPEED_LAG_ERROR;
       #PO.x_Bit_3_deactivate_speed_monitoring := #DEACTIVATE_SPEED_MONITORING;

       //Set the not used Bits to "false"
       #PO.x_Bit_2 := FALSE;
       #PO.x_Bit_4:= FALSE;
       #PO.x_Bit_5:= FALSE;
       #PO.x_Bit_6 := FALSE;
       #PO.x_Bit_7 := FALSE;
       #PO.x_Bit_8 := FALSE;
       #PO.x_Bit_9 := FALSE;
       #PO.x_Bit_10:= FALSE;
       #PO.x_Bit_11:= FALSE;
       #PO.x_Bit_12:= FALSE;
       #PO.x_Bit_13:= FALSE;
       #PO.x_Bit_14:= FALSE;
       #PO.x_Bit_15:= FALSE;

       #PO.i_maximum_torque := #MAXIMUM_TORQUE;

   ELSE
       GOTO END;
   END_IF;

   //DPWR_DAT: Write consistent data of a DP standard slave/PROFINET IO device
   #DPWR_RET_VAL := DPWR_DAT(LADDR := #HW_IDENTIFIER, RECORD := #PO);

   END:
   IF #DPRD_RET_VAL <> 0 OR #DPWR_RET_VAL <> 0 THEN
       #COMMUNICATION_OK := FALSE;

       //Erase FC outputs in case of an error
       #TORQUE_LIMIT_VIA_PD_ACTIVE := FALSE;
       #SPEED_LAG_ERROR_MONITORING_INACTIVE := FALSE;
       #TORQUE_LIMIT_REACHED := FALSE;
       #SPEED_MONITORING_INACTIVE := FALSE;

       #ACTUAL_TORQUE := 0;
   END_IF;
END_FUNCTION

ORGANIZATION_BLOCK "Main"   // OB1, FBD, ProgramCycle
TITLE = "Main Program Sweep (Cycle)"
{ S7_Optimized_Access := 'TRUE' }
VERSION : 0.1
// This sample program only demonstrates the basic approach. We do not accept any legal or other liability for incorrect program functions and their consequences!
// 
// Please take note of the manual "MOVIKIT® Positioning, Velocity"
BEGIN

REGION Network 1: Control of the drive velocity-UDT-S712xx with the functions "Variable jerk time, Variable torque limitation, parameter channel via process data (5PD).
   // Control of the drive velocity-UDT-S712xx with the functions "Variable jerk time, Variable torque limitation, parameter channel via process data (5PD).
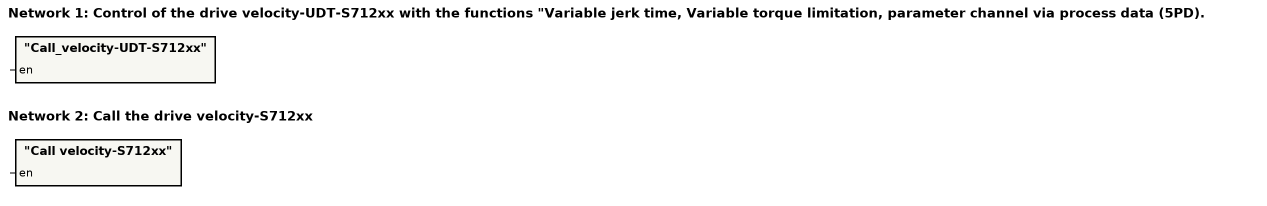
   "Call_velocity-UDT-S712xx"();
END_REGION

REGION Network 2: Call the drive velocity-S712xx
   // without the use of UDTs, without the functions "Variable jerk time, Variable torque limitation, parameter channel via process data (5PD)
   "Call velocity-S712xx"();
END_REGION
END_ORGANIZATION_BLOCK

// folder: 5_PD_Parameter_channel

FUNCTION_BLOCK "5_PD_parameter_channel_FB"   // FB198, SCL
TITLE = 5_PD_parameter_channel_FB
{ S7_Optimized_Access := 'FALSE' }
AUTHOR : SVSPASE
FAMILY : MOVIKIT
VERSION : 2.0
// This sample program only demonstrates the basic approach. We do not accept any legal or other liability for incorrect program functions and their consequences!
// 
// This FB is used to control the MOVIKIT function "parameter channel via process dada (5PD)"
// 
// Device & networks: To use this FB, a 5 PD slot must be configured.
// 
// This FC uses the UDTs "SEW_MOVIKIT_5_PD_PAR_SETPOINTS_V2.0" and "SEW_MOVIKIT_5_PD_PAR_STATUS_V2.0". 
// Please make sure that these PLC data types are available in your TIA project. 
// These UDTs can be copied from the original TIA sample project or from the MOVIKIT_Vel_&_Pos_UDTs_V2.0.al14 library.
// 
// Attention Input "HW_Identifier":
// Assign the HW-Identifier of the 5 PD slot. S73xx/4xx:Change Data type from HW_IO to WORD;  Assign the peripheral address of the 5 PD slot
   VAR_INPUT
      HW_Identifier : Hw_Io;   // S71xxx: Assign the HW-Identifier of the 5 PD slot. S73xx/4xx:Change Data type from HW_IO to WORD; Assign the peripheral address of the 5 PD slot
      SERVICE : Bool;   // false: READ; true: WRITE
      INDEX : Int;   // Index
      SubIndex : Byte;   // Subindex
      OFFSET : Byte;   // Offset
      WRITE_DATA : DWord;   // value to write
   END_VAR
   VAR_OUTPUT
      COMMUNICATION_NOT_OK : Bool;   // true: DPRD_DAT and DPWR_DAT are not working correctly. 5 PD slot required; Check input "HW_Identifier"
      TIMEOUT : Bool;   // true: the participant does not respond.
      READ_SERVICE_SELECTED : Bool;   // "Read" service selected
      WRITE_SERVICE_SELECTED : Bool;   // "Write" service selected
      ERROR : Bool;   // Service failed
      ACTUAL_INDEX : Int;   // selected Index
      ACTUAL_SUBINDEX : Byte;   // selected Subindex
      ACTUAL_OFFSET : Byte;   // selected Offset
      READ_DATA_OR_ERROR_CODE : DWord;   // Read value or error code at Error = true; Error codes are documented in the manual "MOVIKIT POSITIONING VELOCITY DRIVE"
   END_VAR
   VAR_IN_OUT
      ACTIVATE : Bool;   // activate a parameter service
      BUSY : Bool;   // the parameter service is busy right now
      DONE : Bool;   // a parameter service is done
   END_VAR
   VAR
      PI : "SEW_MOVIKIT_5_PD_PAR_STATUS_V2.0";
      PO : "SEW_MOVIKIT_5_PD_PAR_SETPOINTS_V2.0";
      DPRD_RET_VAL : Int;
      DPWR_RET_VAL : Int;
      TimeoutCounter : Int := 1000;
   END_VAR
BEGIN
   (*This sample program only demonstrates the basic approach. We do not accept any legal or other liability for incorrect program functions and their consequences!

   This FB198 serves as a program block for controlling the MOVIKIT function "Parameter channel via process data 5PD)" for the generation C device series,
   Which is implemented up to Movi-C main firmware 9.00.
   Device & networks: To use this FB, a 5 PD slot must be configured.

   This FC uses the UDTs "SEW_MOVIKIT_5_PD_PAR_SETPOINTS_V2.0" and "SEW_MOVIKIT_5_PD_PAR_STATUS_V2.0". 
   Please make sure that these PLC data types are available in your TIA project. 
   These UDTs can be copied from the original TIA sample project or from the MOVIKIT_Vel_&_Pos_UDTs_V2.0.al14 library.

   Attention Input "HW_Identifier":
   Assign the HW-Identifier of the 5 PD slot. S73xx/4xx:Change Data type from HW_IO to WORD;  Assign the peripheral address of the 5 PD slot*)


   IF #ACTIVATE THEN //Initilization
       #ACTIVATE := false; 
       #BUSY := true;
       #DONE := false;
       #TIMEOUT := false;
       #TimeoutCounter := 1000;

   //Assign the POs:
       IF #SERVICE = false THEN //Read service
           #PO.x_Bit_8_READ := true;
           #PO.x_Bit_9_WRITE := false;
       ELSE
           #PO.x_Bit_8_READ:= false;
           #PO.x_Bit_9_WRITE :=true; //Write service
       END_IF;

       #PO.x_Bit_14_execute_function:= false; //Prepare positive signal edge
       #PO.i_Index := #INDEX;
       #PO.b_Offset := #OFFSET;
       #PO.b_SubIndex:= #SubIndex;
       #PO.dw_value:=#WRITE_DATA;

     //Write the init. values: DPWR_DAT: Write consistent data of a DP standard slave/PROFINET IO device
       #DPWR_RET_VAL := DPWR_DAT(LADDR := #HW_Identifier, RECORD := #PO);
      RETURN; // //exit the FB; end of the init. 
   END_IF;


   IF #BUSY = 1 THEN
       //Timeout monitoring
       #TimeoutCounter := #TimeoutCounter - 1;
       IF #TimeoutCounter = 0 THEN
           #ERROR := true;
           #BUSY := false;
           #DONE := true;
           #TIMEOUT := true;
           #READ_DATA_OR_ERROR_CODE := 0;
           RETURN; //exit the FB
       END_IF;


           #DPRD_RET_VAL := DPRD_DAT(LADDR := #HW_Identifier, RECORD => #PI);   //DPRD_DAT: Read consistent data of a DP standard slave
           IF #DPRD_RET_VAL = 0 THEN
               #COMMUNICATION_NOT_OK := 0; 

               IF #INDEX = #PI.i_actual_Index THEN                 //Check whether the parameter channel already reports back the sent data           
                   #PO.x_Bit_14_execute_function := true;  

                   IF #PI.x_Bit_14_Service_completed = true THEN  //If "Service is completed" the parameter service is "done"..
                               #BUSY := false;
                               #DONE := true;

                   END_IF;
     //Mapping of the process input data   
                   #READ_SERVICE_SELECTED := #PI.x_Bit_8_READ_Service_selected;
                   #WRITE_SERVICE_SELECTED := #PI.x_Bit_9_WRITE_Service_selected;
                   #ERROR := #PI.x_Bit_15_Service_failed;
                   #ACTUAL_INDEX := #PI.i_actual_Index;
                   #ACTUAL_OFFSET := #PI.b_actual_Offset; //WORD_TO_INT(#PI[3] AND w#16#ff);//Hide the high-byte
                   #ACTUAL_SUBINDEX := #PI.b_actual_SubIndex;//WORD_TO_INT(SHR(IN := #PI[3], N := 8)); //shift 8 Bits/1 Byte right...
                   #READ_DATA_OR_ERROR_CODE := #PI.dw_value_read;
       END_IF;

       #DPWR_RET_VAL := DPWR_DAT(LADDR := #HW_Identifier, RECORD := #PO); //DPWR_DAT: Write consistent data of a DP standard slave/PROFINET IO device

       ELSE
           GOTO END;
       END_IF; 

       END:
       IF #DPRD_RET_VAL <> 0 OR #DPWR_RET_VAL <> 0  THEN
               #BUSY := false;
               #DONE := true;
               #ERROR := true;
               #COMMUNICATION_NOT_OK := 1;
               //Erase FB outputs in case of an error
               #READ_SERVICE_SELECTED := false;
               #WRITE_SERVICE_SELECTED := false;
               #ACTUAL_INDEX := 0;
               #ACTUAL_SUBINDEX := 0;
               #ACTUAL_OFFSET := 0;
               #READ_DATA_OR_ERROR_CODE := 0;
           END_IF;
       END_IF;  //Busy
END_FUNCTION_BLOCK

FUNCTION "Call velocity-UDT-S712xx_parameter channel via process data (5PD)" : Void   // FC105, FBD
TITLE = Call 5 PD Parameter channel
{ S7_Optimized_Access := 'TRUE' }
VERSION : 0.1
// This sample program only demonstrates the basic approach. We do not accept any legal or other liability for incorrect program functions and their consequences!
// 
// This FB198 serves as a program block for controlling the MOVIKIT function "Parameter channel via process data 5PD)" for the generation C device series,
// which is implemented up to Movi-C main firmware 9.00.
// Device & networks: To use this FB, a 5 PD slot must be configured.
BEGIN

REGION Network 1: Slot 5; Reading the head sink temperature - Mapping of Index & SubIndex
   // MoviSuite: Diagnostics/Process values/Output stage/Utilization/Heat sink temperature; 
   // Index 8312; SubIndex 5
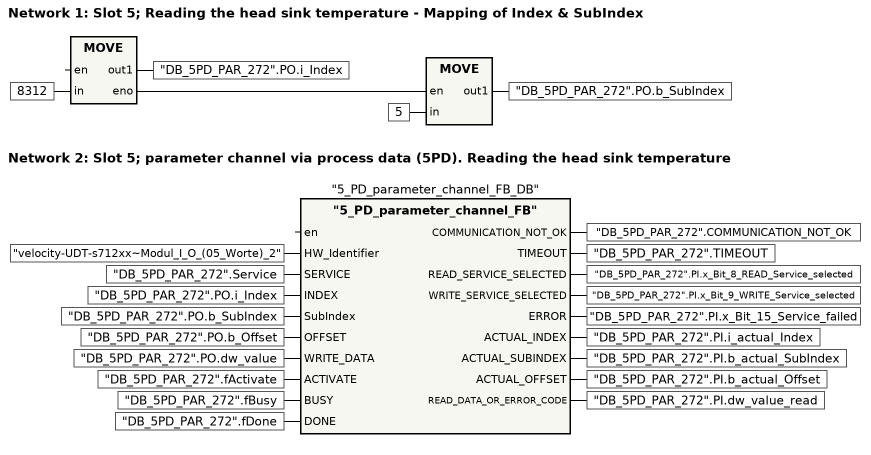
   // ENO of a box is taken as its EN; it also drops when the box reports an error
   "DB_5PD_PAR_272".PO.i_Index := 8312;
   "DB_5PD_PAR_272".PO.b_SubIndex := 5;
END_REGION

REGION Network 2: Slot 5; parameter channel via process data (5PD). Reading the head sink temperature
   // MoviSuite: Diagnostics/Process values/Output stage/Utilization/Heat sink temperature; 
   // Index 8312; SubIndex 5 
   // 
   // With this additional function, parameters can be read and written volatile.
   // The Additional function extends the process data length by 5 process data words.
   // 
   // Inputs of the FB:
   // 
   // Attention! 
   // S71xxx: "HW_Identifier". Assign the HW-Identifier of the 5 PD slot. 
   // S73xx/4xx:"HW_Identifier"Change the data type from "HW_IO" to "WORD" Assign the peripheral address of the 5 PD slot;
   // 
   // "SERVICE": false: READ; true: WRITE
   // "INDEX": Index
   // "SubIndex": Subindex
   // "OFFSET": Offset
   // "WRITE_DATA": value to write
   // 
   // 
   // Outputs of the FB:
   // 
   // "COMMUNICATION_NOT_OK": true: DPRD_DAT and DPWR_DAT are not working correctly. 5 PD slot required; 
   //                                                    Check input  "HW_Identifier"
   // "TIMEOUT": true: true:  the participant does not respond.
   // "READ_SERVICE_SELECTED": "Read" service selected
   // "WRITE_SERVICE_SELECTED": "Write" service selected
   // "ERROR": Service failed
   // "ACTUAL_INDEX": selected Index
   // "ACTUAL_SUBINDEX": selected Subindex
   // "ACTUAL_OFFSET": selected Offset
   // "READ_DATA_OR_ERROR_CODE": Read value or error code at Error = true; Error codes are documented in the manual                                                           "MOVIKIT POSITIONING VELOCITY DRIVE"
   // 
   // Status machine of the FB:
   // ACTIVATE: activate a parameter service
   // BUSY: the parameter service is busy right now
   // DONE: a parameter service is done
   "5_PD_parameter_channel_FB_DB"(HW_Identifier := "velocity-UDT-s712xx~Modul_I_O_(05_Worte)_2",   // "5_PD_parameter_channel_FB"
                           SERVICE := "DB_5PD_PAR_272".Service,
                           INDEX := "DB_5PD_PAR_272".PO.i_Index,
                           SubIndex := "DB_5PD_PAR_272".PO.b_SubIndex,
                           OFFSET := "DB_5PD_PAR_272".PO.b_Offset,
                           WRITE_DATA := "DB_5PD_PAR_272".PO.dw_value,
                           ACTIVATE := "DB_5PD_PAR_272".fActivate,
                           BUSY := "DB_5PD_PAR_272".fBusy,
                           DONE := "DB_5PD_PAR_272".fDone,
                           COMMUNICATION_NOT_OK => "DB_5PD_PAR_272".COMMUNICATION_NOT_OK,
                           TIMEOUT => "DB_5PD_PAR_272".TIMEOUT,
                           READ_SERVICE_SELECTED => "DB_5PD_PAR_272".PI.x_Bit_8_READ_Service_selected,
                           WRITE_SERVICE_SELECTED => "DB_5PD_PAR_272".PI.x_Bit_9_WRITE_Service_selected,
                           ERROR => "DB_5PD_PAR_272".PI.x_Bit_15_Service_failed,
                           ACTUAL_INDEX => "DB_5PD_PAR_272".PI.i_actual_Index,
                           ACTUAL_SUBINDEX => "DB_5PD_PAR_272".PI.b_actual_SubIndex,
                           ACTUAL_OFFSET => "DB_5PD_PAR_272".PI.b_actual_Offset,
                           READ_DATA_OR_ERROR_CODE => "DB_5PD_PAR_272".PI.dw_value_read);
END_REGION
END_FUNCTION

// ===== PLC "CPU 315F-2 PN/DP"  CPU 315F-2 PN/DP =====

VAR_GLOBAL   // PLC tag table "Standard-Variablentabelle"
   "Clock_0.5Hz" AT %M0.7 : Bool;
   "Clock_Byte" AT %MB0 : Byte;
   "Clock_10Hz" AT %M0.0 : Bool;
   "Clock_5Hz" AT %M0.1 : Bool;
   "Clock_2.5Hz" AT %M0.2 : Bool;
   "Clock_2Hz" AT %M0.3 : Bool;
   "Clock_1.25Hz" AT %M0.4 : Bool;
   "Clock_1Hz" AT %M0.5 : Bool;
   "Clock_0.625Hz" AT %M0.6 : Bool;
   "velocity-UDT-S73xx_PO1" AT %AW300 : Word;   // control word
   "velocity-UDT-S73xx_PO2" AT %QW302 : Word;   // setpoint speed
   "velocity-UDT-S73xx_PO3" AT %QW304 : Word;   // acceleration
   "velocity-UDT-S73xx_PO4" AT %QW306 : Word;   // deceleration
   "velocity-UDT-S73xx_PO5" AT %QW308 : Word;   // dig. Outputs
   "velocity-UDT-S73xx_PI1" AT %IW300 : Word;   // status word
   "velocity-UDT-S73xx_PI2" AT %IW302 : Word;   // actual speed
   "velocity-UDT-S73xx_PI3" AT %IW304 : Word;   // Status/Main/Subfault
   "velocity-UDT-S73xx_PI4" AT %IW306 : Word;   // actual torque
   "velocity-UDT-S73xx_PI5" AT %IW308 : Word;   // dig. Inputs
END_VAR

TYPE "SEW_MOVIKIT_VelocityDrive_STATUS_V2.1"
// Dieses UDT bildet die 5 Prozeßausgangsdaten des MOVIKIT VelocityDrives ab. This UDT maps the 5 process output data of the MOVIKIT VelocityDrive.
   STRUCT
      x_Bit_8_Fault : Bool;
      x_Bit_9_Warning : Bool;
      x_Bit_10_DriveTrain2_active : Bool;
      x_Bit_11_Setp_actual_speed_comp_signal_active : Bool;
      x_Bit_12_SW_Limit_switches_inactive : Bool;
      x_Bit_13_Reserved : Bool;
      x_Bit_14_StandBy_Mode_active : Bool;
      x_Bit_15_Heartbeat_OUT : Bool;
      x_Bit_0_Ready : Bool;
      x_Bit_1_STO_inactive : Bool;
      x_Bit_2_Output_Stage_enabled : Bool;
      x_Bit_3_Brake_released : Bool;
      x_Bit_4_Motor_turning : Bool;
      x_Bit_5_Active_Drive_referenced : Bool;
      x_Bit_6_New_Relative_Position_applied : Bool;
      x_Bit_7_In_Position : Bool;
      iActual_Speed : Int;
      wStatus_main_fault_sub_fault : Word;
      iActual_Torque : Int;
      wDigital_Inputs : Word;
   END_STRUCT;
END_TYPE

TYPE "SEW_MOVIKIT_VelocityDrive_SETPOINTS_V2.1"
TITLE = SEW_MOVIKIT_VelocityDrive_SETPOINTS
// Dieses UDT bildet die 5 Prozeßeingangsdaten des MOVIKIT VelocityDrives ab. This UDT maps the 5 process input data of the MOVIKIT VelocityDrive.
   STRUCT
      x_Bit_8_Fault_Reset : Bool;
      x_Bit_9_Reserved : Bool;
      x_Bit_10_Activate_DriveTrain2 : Bool;
      x_Bit_11_Reserved : Bool;
      x_Bit_12_Deactivate_SW_Limit_switches : Bool;
      x_Bit_13_Activate_Output_Stage_Inhibit : Bool;
      x_Bit_14_Activate_StandBy : Bool;
      x_Bit_15_Heartbeat_IN : Bool;
      x_Bit_0_Enable_Emergency_Stop : Bool;
      x_Bit_1_Enable_Application_Stop : Bool;
      x_Bit_2_Reserved : Bool;
      x_Bit_3_Release_Brake : Bool;
      x_Bit_4_Jog_positive : Bool;
      x_Bit_5_Jog_negative : Bool;
      x_Bit_6_Apply_relative_Position : Bool;
      x_Bit_7_Start_Stop : Bool;
      iSetpoint_Speed : Int;
      iAcceleration : Int;
      iDeceleration : Int;
      wDigital_Outputs : Word;
   END_STRUCT;
END_TYPE

DATA_BLOCK "MOVIKIT_Velocity_256"   // DB256
{ S7_Optimized_Access := 'FALSE' }
VERSION : 0.1
   VAR
      PO : "SEW_MOVIKIT_VelocityDrive_SETPOINTS_V2.1";
      PI : "SEW_MOVIKIT_VelocityDrive_STATUS_V2.1";
      Communication_OK : Bool;   // true: DPRD_DAT and DPWR_DAT are working correctly. false: 5 PD slot required; Check address at Input "IO_ADDRESS"
   END_VAR
BEGIN
END_DATA_BLOCK

FUNCTION "Call_Velocity_UDT_S73xx" : Void   // FC100, FBD
TITLE = Call_Velocity_UDT_S73xx
{ S7_Optimized_Access := 'FALSE' }
VERSION : 0.1
// This sample program only demonstrates the basic approach. We do not accept any legal or other liability for incorrect program functions and their consequences!
// 
// Please take note of the manual "MOVIKIT® Positioning, Velocity"
BEGIN

REGION Network 1: Control of the drive velocity-UDT-S73xx
   // The FC122 serves as a program module for controlling the MOVIKIT module "Velocity Drive" for the Generation C device series. With the help of the FC122, the converters can be controlled via PROFINET IO/PROFIBUS DP. 
   // 
   // Device & networks: To use this FC, a 5 PD slot must be configured.
   // 
   // This FC uses the UDTs "SEW_MOVIKIT_VelocityDrive_SETPOINTS_V2.1" and "SEW_MOVIKIT_VelocityDrive_STATUS_V2.1". Please make sure that these PLC data types are available in your TIA project. These UDTs can be copied from the original TIA sample project or from the MOVIKIT_Vel_&_Pos_UDTs_V2.x.al14 library.
   // 
   // Inputs of the FC:
   // 
   // Attention! 
   // S73xx/4xx:"IO_ADDRESS"/Data Type Word:  Assign the peripheral address of the 5 PD slot;
   // S71xxx: "IO_ADDRESS" change the data type from Word to "HW_IO". Assign the HW-Identifier of the 5 PD slot. 
   // 
   // "ENABLE_EMERGENCY_STOP" = true: Enable; false: emergency stop
   // "ENABLE_APPLICATION_STOP" = true: Enable; false: Application stop
   // "RELEASE_BRAKE" = true: release brake (without enable)
   // "START_STOP" = Start/stop with fieldbus ramp
   // "FAULT_RESET": true: Fault reset
   // "ACTIVATE_DRIVE_TRAIN_2" = true: Activate drive train 2
   // "ACTIVATE_OUPUT_STAGE_INHIBIT" = true: Activate output stage inhibit
   // "ACTIVATE_STANDBY_MODE" = true: Activate standby mode
   // "HEARTBEAT_IN": Copied to "HEARTBEAT_OUT"
   // "SETPOINT_SPEED": in user unit (INT) 
   // "SETPOINT_ACCELERATION":  in user unit (INT) 
   // "SETPOINT_DECELERATION":  in user unit (INT)
   // "DIGITAL_OUTPUTS": MoviSuite/Movikit../Inputs/Outputs: dig Outputs: the setting "control via fieldbus" is needed
   // 
   // Outputs of the FC:
   // 
   // If the data transmission/PROFINET is disrupted, all outputs will be deleted..
   // => "COMMUNICATION_OK = false (self-confirming)
   // "READY" = true: Ready for operation.
   // "STO_INACTIVE" = true: STO inactive.
   // "OUTPUT_STAGE_ENABLED" = true: Output stage enabled.
   // "BRAKE_RELEASED" = true: Brake released.
   // "MOTOR_TURNING" = true: Motor turning.
   // "FAULT" = true: Fault.
   // "WARNING" = true: Warning 
   // "DRIVE_TRAIN_2_ACTIVE" = true: Drive train 2 active.
   // "SETPOINT-ACTUAL_COMPARISON" 
   // "STANDBY_MODE_ACTIVE" = true: Stand-by Mode is active.
   // "HEARTBEAT_OUT" : This signal is copied internally from "HEARTBEAT_IN"
   // "ACTUAL_SPEED": in user unit (INT) 
   // "STATUS_MAIN_FAULT_SUB_FAULT:" (WORD)
   //    No fault: Display of current FCB; fault/warning:  High-Byte Fault; Low-Byte SubFault
   // "ACTUAL_TORQUE":in user unit (INT)
   // "DIGITAL_INPUTS" : The digital inputs are read out
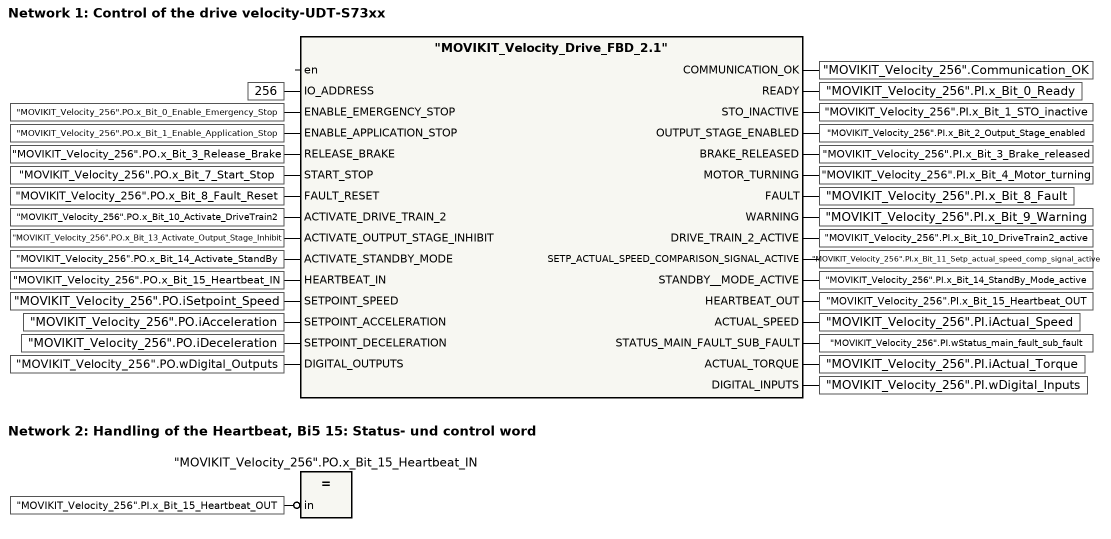
   "MOVIKIT_Velocity_Drive_FBD_2.1"(IO_ADDRESS := 256,
                           ENABLE_EMERGENCY_STOP := "MOVIKIT_Velocity_256".PO.x_Bit_0_Enable_Emergency_Stop,
                           ENABLE_APPLICATION_STOP := "MOVIKIT_Velocity_256".PO.x_Bit_1_Enable_Application_Stop,
                           RELEASE_BRAKE := "MOVIKIT_Velocity_256".PO.x_Bit_3_Release_Brake,
                           START_STOP := "MOVIKIT_Velocity_256".PO.x_Bit_7_Start_Stop,
                           FAULT_RESET := "MOVIKIT_Velocity_256".PO.x_Bit_8_Fault_Reset,
                           ACTIVATE_DRIVE_TRAIN_2 := "MOVIKIT_Velocity_256".PO.x_Bit_10_Activate_DriveTrain2,
                           ACTIVATE_OUTPUT_STAGE_INHIBIT := "MOVIKIT_Velocity_256".PO.x_Bit_13_Activate_Output_Stage_Inhibit,
                           ACTIVATE_STANDBY_MODE := "MOVIKIT_Velocity_256".PO.x_Bit_14_Activate_StandBy,
                           HEARTBEAT_IN := "MOVIKIT_Velocity_256".PO.x_Bit_15_Heartbeat_IN,
                           SETPOINT_SPEED := "MOVIKIT_Velocity_256".PO.iSetpoint_Speed,
                           SETPOINT_ACCELERATION := "MOVIKIT_Velocity_256".PO.iAcceleration,
                           SETPOINT_DECELERATION := "MOVIKIT_Velocity_256".PO.iDeceleration,
                           DIGITAL_OUTPUTS := "MOVIKIT_Velocity_256".PO.wDigital_Outputs,
                           COMMUNICATION_OK => "MOVIKIT_Velocity_256".Communication_OK,
                           READY => "MOVIKIT_Velocity_256".PI.x_Bit_0_Ready,
                           STO_INACTIVE => "MOVIKIT_Velocity_256".PI.x_Bit_1_STO_inactive,
                           OUTPUT_STAGE_ENABLED => "MOVIKIT_Velocity_256".PI.x_Bit_2_Output_Stage_enabled,
                           BRAKE_RELEASED => "MOVIKIT_Velocity_256".PI.x_Bit_3_Brake_released,
                           MOTOR_TURNING => "MOVIKIT_Velocity_256".PI.x_Bit_4_Motor_turning,
                           FAULT => "MOVIKIT_Velocity_256".PI.x_Bit_8_Fault,
                           WARNING => "MOVIKIT_Velocity_256".PI.x_Bit_9_Warning,
                           DRIVE_TRAIN_2_ACTIVE => "MOVIKIT_Velocity_256".PI.x_Bit_10_DriveTrain2_active,
                           SETP_ACTUAL_SPEED_COMPARISON_SIGNAL_ACTIVE => "MOVIKIT_Velocity_256".PI.x_Bit_11_Setp_actual_speed_comp_signal_active,
                           STANDBY__MODE_ACTIVE => "MOVIKIT_Velocity_256".PI.x_Bit_14_StandBy_Mode_active,
                           HEARTBEAT_OUT => "MOVIKIT_Velocity_256".PI.x_Bit_15_Heartbeat_OUT,
                           ACTUAL_SPEED => "MOVIKIT_Velocity_256".PI.iActual_Speed,
                           STATUS_MAIN_FAULT_SUB_FAULT => "MOVIKIT_Velocity_256".PI.wStatus_main_fault_sub_fault,
                           ACTUAL_TORQUE => "MOVIKIT_Velocity_256".PI.iActual_Torque,
                           DIGITAL_INPUTS => "MOVIKIT_Velocity_256".PI.wDigital_Inputs);
END_REGION

REGION Network 2: Handling of the Heartbeat, Bi5 15: Status- und control word
   "MOVIKIT_Velocity_256".PO.x_Bit_15_Heartbeat_IN := NOT "MOVIKIT_Velocity_256".PI.x_Bit_15_Heartbeat_OUT;
END_REGION
END_FUNCTION

FUNCTION "MOVIKIT_Velocity_Drive_FBD_2.1" : Void   // FC122, FBD
TITLE = MOVIKIT Velocity Drive/S73xx in FBD_2.1
{ S7_Optimized_Access := 'FALSE' }
AUTHOR : CSCEASDI
FAMILY : MOVIKIT
VERSION : 2.1
// This sample program only demonstrates the basic approach. We do not accept any legal or other liability for incorrect program functions and their consequences!
// 
// The FC122 serves as a program module for controlling the MOVIKIT module "Velocity Drive" for the Generation C device series. With the help of the FC122, the converters can be controlled via PROFINET IO/PROFIBUS DP. 
// 
// Device & networks: To use this FC, a 5 PD slot must be configured.
// 
// This FC uses the UDTs SEW_MOVIKIT_VelocityDrive_SETPOINTS_V2.0 and SEW_MOVIKIT_VelocityDrive_STATUS_V2.0. Please make sure that these PLC data types are available in your TIA project. These UDTs can be copied from the original TIA sample project or from the MOVIKIT_Vel_&_Pos_UDTs_V2.0.al14 library.
// 
// Attention! 
// S73xx/4xx:"IO_ADDRESS"/Data Type Word:  Assign the peripheral address of the 5 PD slot;
// S71xxx: "IO_ADDRESS" change the data type from Word to "HW_IO". Assign the HW-Identifier of the 5 PD slot.
   VAR_INPUT
      IO_ADDRESS : Word;   // S73xx/4xx:"IO_ADDRESS"/Data Type Word: Assign the peripheral address of the 5 PD slot; S71xxx: "IO_ADDRESS" change the data type from Word to "HW_IO". Assign the HW-Identifier of the 5 PD slot.
      ENABLE_EMERGENCY_STOP : Bool;   // true: Enable; false: emergency stop
      ENABLE_APPLICATION_STOP : Bool;   // true: Enable; false: Application stop
      RELEASE_BRAKE : Bool;   // true: release brake (without enable)
      START_STOP : Bool;   // Start/stop with fieldbus ramp
      FAULT_RESET : Bool;   // true: Fault reset
      ACTIVATE_DRIVE_TRAIN_2 : Bool;   // true: Activate drive train 2
      ACTIVATE_OUTPUT_STAGE_INHIBIT : Bool;   // true: Activate output stage inhibit
      ACTIVATE_STANDBY_MODE : Bool;   // true: Activate standby mode
      HEARTBEAT_IN : Bool;   // Copied to "HEARTBEAT_OUT"
      SETPOINT_SPEED : Int;   // in user unit (INT)
      SETPOINT_ACCELERATION : Int;   // in user unit (INT)
      SETPOINT_DECELERATION : Int;   // in user unit (INT)
      DIGITAL_OUTPUTS : Word;   // MoviSuite/Movikit../Inputs/Outputs: dig Outputs: the setting "control via fieldbus" is needed
   END_VAR
   VAR_OUTPUT
      COMMUNICATION_OK : Bool;   // true: DPRD_DAT and DPWR_DAT are working correctly. false: 5 PD slot required; Check address at Input "IO_ADDRESS"
      READY : Bool;   // true: Ready for operation.
      STO_INACTIVE : Bool;   // true: STO inactive.
      OUTPUT_STAGE_ENABLED : Bool;   // true: Output stage enabled.
      BRAKE_RELEASED : Bool;   // true: Brake released.
      MOTOR_TURNING : Bool;   // true: Motor turning.
      FAULT : Bool;   // true: Fault.
      WARNING : Bool;   // true: Warning
      DRIVE_TRAIN_2_ACTIVE : Bool;   // true: Drive train 2 active.
      SETP_ACTUAL_SPEED_COMPARISON_SIGNAL_ACTIVE : Bool;
      STANDBY__MODE_ACTIVE : Bool;   // true: Stand-by Mode is active.
      HEARTBEAT_OUT : Bool;   // This signal is copied internally from "HEARTBEAT_IN"
      ACTUAL_SPEED : Int;   // in user unit (INT)
      STATUS_MAIN_FAULT_SUB_FAULT : Word;   // No fault: Display of current FCB; fault/warning: High-Byte Fault; Low-Byte SubFault
      ACTUAL_TORQUE : Int;   // in user unit (INT)
      DIGITAL_INPUTS : Word;   // The digital inputs are read out
   END_VAR
   VAR_TEMP
      PI : "SEW_MOVIKIT_VelocityDrive_STATUS_V2.1";   // Dieses UDT bildet die 5 Prozeßeingangsdaten des MOVIKIT VelocityDrives ab. This UDT maps the 5 process input data of the MOVIKIT VelocityDrive.
      PO : "SEW_MOVIKIT_VelocityDrive_SETPOINTS_V2.1";   // Dieses UDT bildet die 5 Prozeßausgangsdaten des MOVIKIT VelocityDrives ab. This UDT maps the 5 process output data of the MOVIKIT VelocityDrive.
      DPRD_RET_VAL : Int;
      DPWR_RET_VAL : Int;
      Com_DPRD_OK : Bool;
      Com_DPWR_OK : Bool;
      FALSE : Bool;
   END_VAR
   VAR_TEMP   // added for the SCL form of the ladder/FBD networks
      _w1 : Bool;
   END_VAR
BEGIN

REGION Network 1: Def."#FALSE"
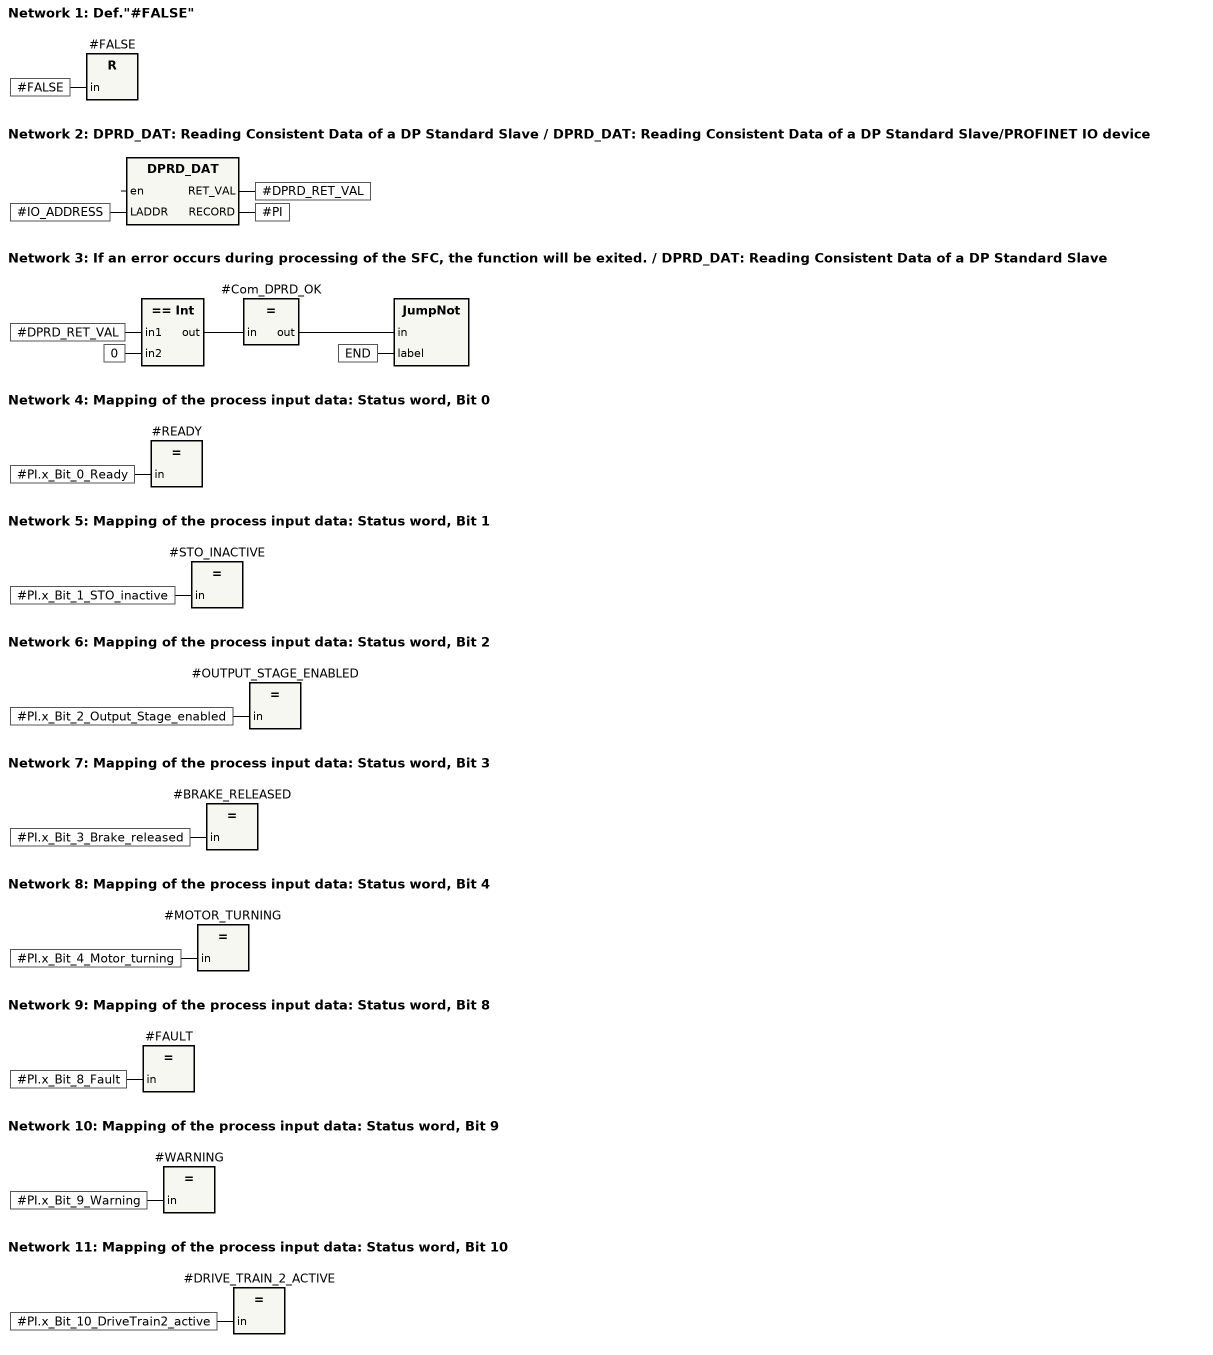
   IF #FALSE THEN #FALSE := FALSE; END_IF;
END_REGION

REGION Network 2: DPRD_DAT: Reading Consistent Data of a DP Standard Slave / DPRD_DAT: Reading Consistent Data of a DP Standard Slave/PROFINET IO device
   #DPRD_RET_VAL := DPRD_DAT(LADDR := #IO_ADDRESS, RECORD => #PI);
END_REGION

REGION Network 3: If an error occurs during processing of the SFC, the function will be exited. / DPRD_DAT: Reading Consistent Data of a DP Standard Slave
   // If the return value = 0, COM_DPRD_OK = TRUE. The function is further processed and not jumped to "END".
   // no SCL statement known for JumpNot: written as a call
   #Com_DPRD_OK := #DPRD_RET_VAL = 0;
   JumpNot(in := #Com_DPRD_OK, label := END);
END_REGION

REGION Network 4: Mapping of the process input data: Status word, Bit 0
   #READY := #PI.x_Bit_0_Ready;
END_REGION

REGION Network 5: Mapping of the process input data: Status word, Bit 1
   #STO_INACTIVE := #PI.x_Bit_1_STO_inactive;
END_REGION

REGION Network 6: Mapping of the process input data: Status word, Bit 2
   #OUTPUT_STAGE_ENABLED := #PI.x_Bit_2_Output_Stage_enabled;
END_REGION

REGION Network 7: Mapping of the process input data: Status word, Bit 3
   #BRAKE_RELEASED := #PI.x_Bit_3_Brake_released;
END_REGION

REGION Network 8: Mapping of the process input data: Status word, Bit 4
   #MOTOR_TURNING := #PI.x_Bit_4_Motor_turning;
END_REGION

REGION Network 9: Mapping of the process input data: Status word, Bit 8
   #FAULT := #PI.x_Bit_8_Fault;
END_REGION

REGION Network 10: Mapping of the process input data: Status word, Bit 9
   #WARNING := #PI.x_Bit_9_Warning;
END_REGION

REGION Network 11: Mapping of the process input data: Status word, Bit 10
   #DRIVE_TRAIN_2_ACTIVE := #PI.x_Bit_10_DriveTrain2_active;
END_REGION

REGION Network 12: Mapping of the process input data: Status word, Bit 11
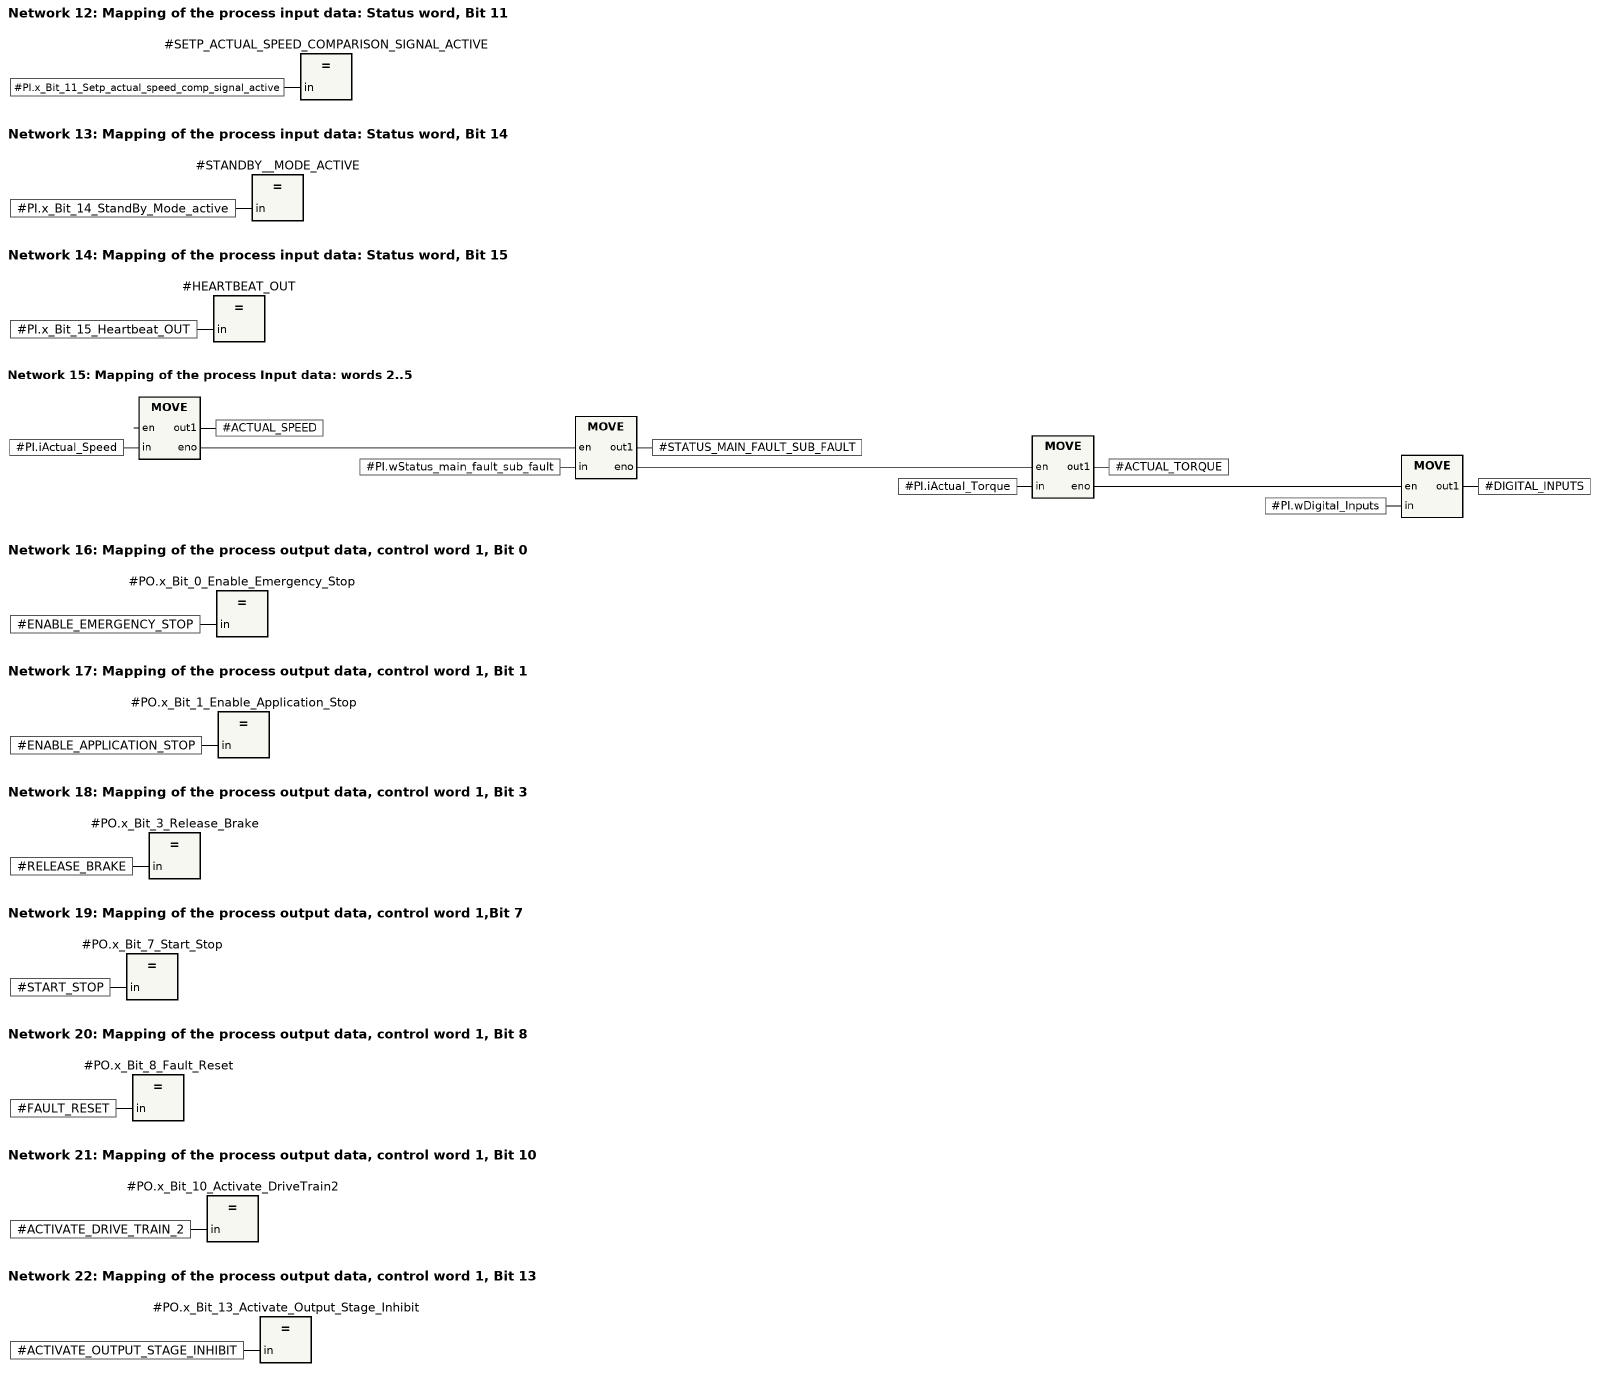
   #SETP_ACTUAL_SPEED_COMPARISON_SIGNAL_ACTIVE := #PI.x_Bit_11_Setp_actual_speed_comp_signal_active;
END_REGION

REGION Network 13: Mapping of the process input data: Status word, Bit 14
   #STANDBY__MODE_ACTIVE := #PI.x_Bit_14_StandBy_Mode_active;
END_REGION

REGION Network 14: Mapping of the process input data: Status word, Bit 15
   #HEARTBEAT_OUT := #PI.x_Bit_15_Heartbeat_OUT;
END_REGION

REGION Network 15: Mapping of the process Input data: words 2..5
   // ENO of a box is taken as its EN; it also drops when the box reports an error
   #ACTUAL_SPEED := #PI.iActual_Speed;
   #STATUS_MAIN_FAULT_SUB_FAULT := #PI.wStatus_main_fault_sub_fault;
   #ACTUAL_TORQUE := #PI.iActual_Torque;
   #DIGITAL_INPUTS := #PI.wDigital_Inputs;
END_REGION

REGION Network 16: Mapping of the process output data, control word 1, Bit 0
   #PO.x_Bit_0_Enable_Emergency_Stop := #ENABLE_EMERGENCY_STOP;
END_REGION

REGION Network 17: Mapping of the process output data, control word 1, Bit 1
   #PO.x_Bit_1_Enable_Application_Stop := #ENABLE_APPLICATION_STOP;
END_REGION

REGION Network 18: Mapping of the process output data, control word 1, Bit 3
   #PO.x_Bit_3_Release_Brake := #RELEASE_BRAKE;
END_REGION

REGION Network 19: Mapping of the process output data, control word 1,Bit 7
   #PO.x_Bit_7_Start_Stop := #START_STOP;
END_REGION

REGION Network 20: Mapping of the process output data, control word 1, Bit 8
   #PO.x_Bit_8_Fault_Reset := #FAULT_RESET;
END_REGION

REGION Network 21: Mapping of the process output data, control word 1, Bit 10
   #PO.x_Bit_10_Activate_DriveTrain2 := #ACTIVATE_DRIVE_TRAIN_2;
END_REGION

REGION Network 22: Mapping of the process output data, control word 1, Bit 13
   #PO.x_Bit_13_Activate_Output_Stage_Inhibit := #ACTIVATE_OUTPUT_STAGE_INHIBIT;
END_REGION

REGION Network 23: Mapping of the process output data, control word 1, Bit 14
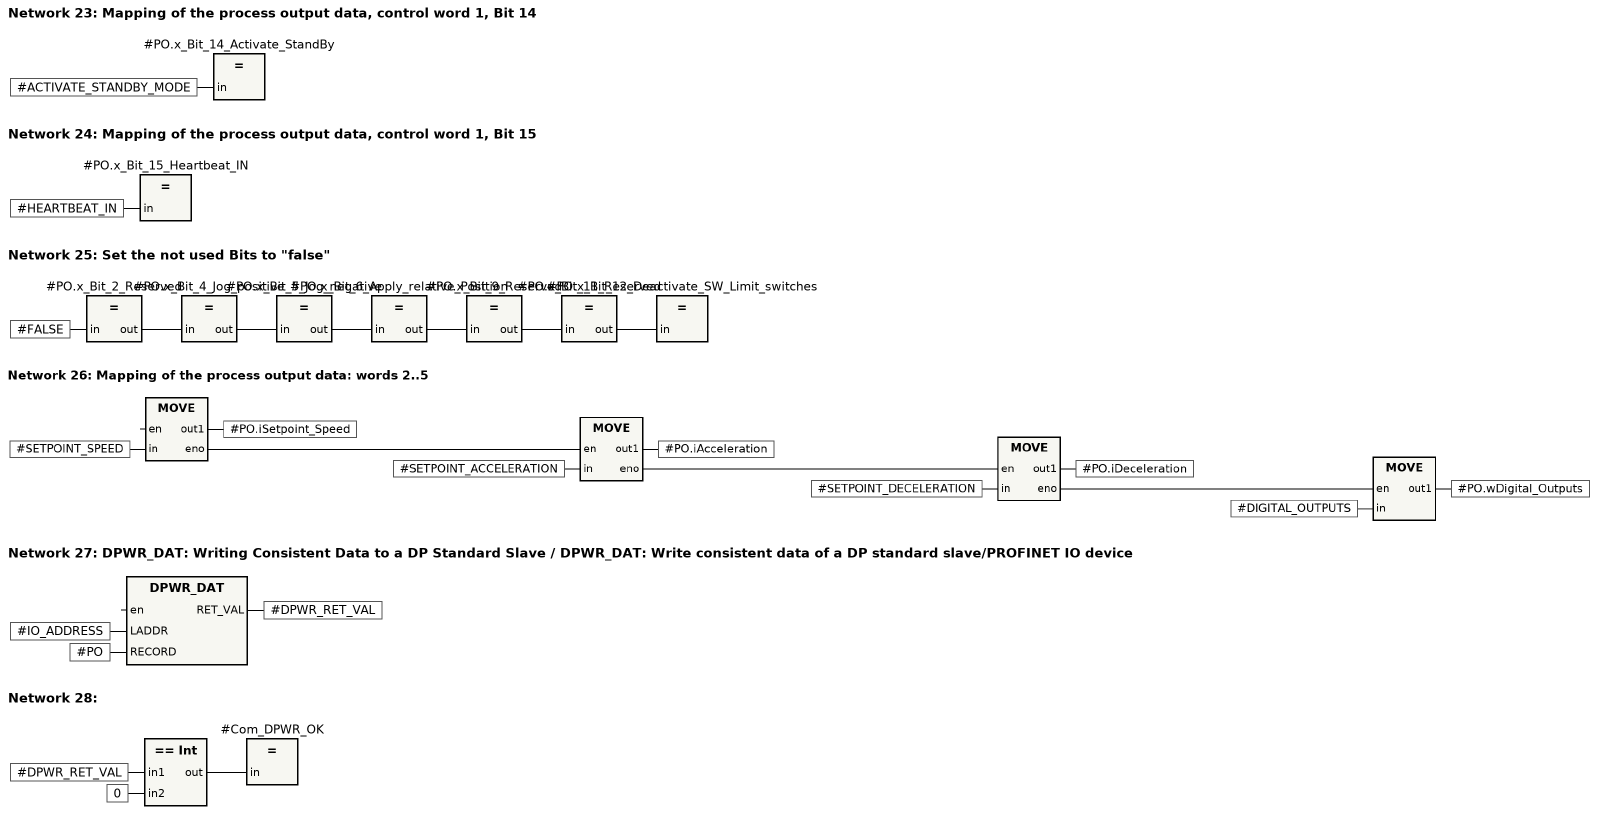
   #PO.x_Bit_14_Activate_StandBy := #ACTIVATE_STANDBY_MODE;
END_REGION

REGION Network 24: Mapping of the process output data, control word 1, Bit 15
   #PO.x_Bit_15_Heartbeat_IN := #HEARTBEAT_IN;
END_REGION

REGION Network 25: Set the not used Bits to "false"
   #PO.x_Bit_2_Reserved := #FALSE;
   #PO.x_Bit_4_Jog_positive := #FALSE;
   #PO.x_Bit_5_Jog_negative := #FALSE;
   #PO.x_Bit_6_Apply_relative_Position := #FALSE;
   #PO.x_Bit_9_Reserved := #FALSE;
   #PO.x_Bit_11_Reserved := #FALSE;
   #PO.x_Bit_12_Deactivate_SW_Limit_switches := #FALSE;
END_REGION

REGION Network 26: Mapping of the process output data: words 2..5
   // ENO of a box is taken as its EN; it also drops when the box reports an error
   #PO.iSetpoint_Speed := #SETPOINT_SPEED;
   #PO.iAcceleration := #SETPOINT_ACCELERATION;
   #PO.iDeceleration := #SETPOINT_DECELERATION;
   #PO.wDigital_Outputs := #DIGITAL_OUTPUTS;
END_REGION

REGION Network 27: DPWR_DAT: Writing Consistent Data to a DP Standard Slave / DPWR_DAT: Write consistent data of a DP standard slave/PROFINET IO device
   // If the DPWR_DAT is processed without errors, the process output data is written consistently. If RET_VAL <> is 0, then there is an error.
   #DPWR_RET_VAL := DPWR_DAT(LADDR := #IO_ADDRESS, RECORD := #PO);
END_REGION

REGION Network 28
   // If the return value = 0, COM_DPWR_OK = TRUE.
   #Com_DPWR_OK := #DPWR_RET_VAL = 0;
END_REGION

REGION Network 29: If processing of SFCs is faulty, all outputs of function will be deleted / Erase FC outputs in case of an error
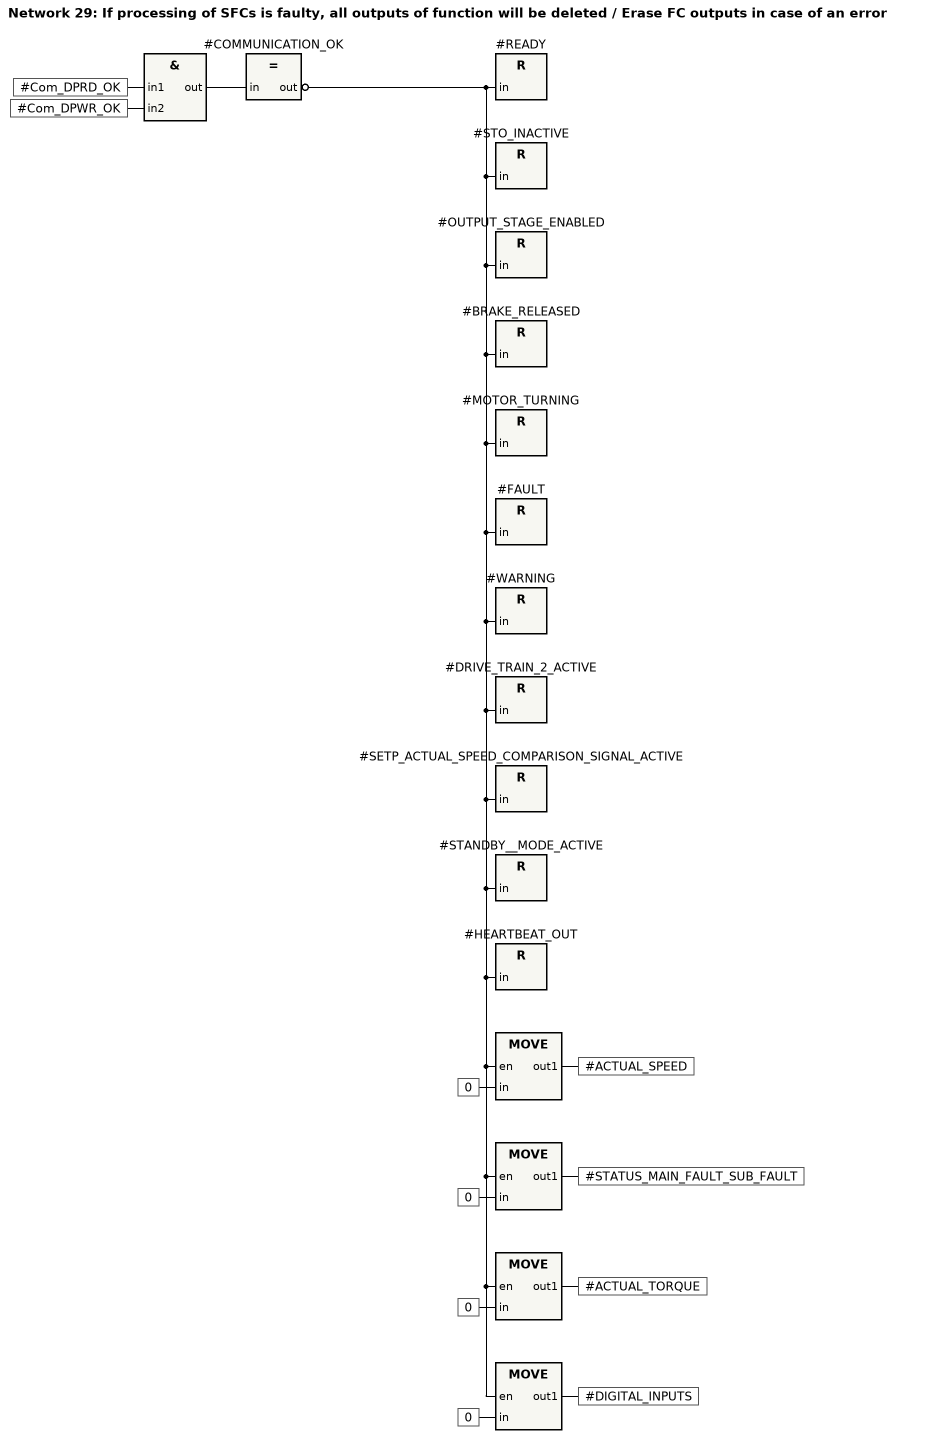
   END:
   #_w1 := #Com_DPRD_OK AND #Com_DPWR_OK;
   #COMMUNICATION_OK := #_w1;
   IF NOT #_w1 THEN
       #READY := FALSE;
       #STO_INACTIVE := FALSE;
       #OUTPUT_STAGE_ENABLED := FALSE;
       #BRAKE_RELEASED := FALSE;
       #MOTOR_TURNING := FALSE;
       #FAULT := FALSE;
       #WARNING := FALSE;
       #DRIVE_TRAIN_2_ACTIVE := FALSE;
       #SETP_ACTUAL_SPEED_COMPARISON_SIGNAL_ACTIVE := FALSE;
       #STANDBY__MODE_ACTIVE := FALSE;
       #HEARTBEAT_OUT := FALSE;
       #ACTUAL_SPEED := 0;
       #STATUS_MAIN_FAULT_SUB_FAULT := 0;
       #ACTUAL_TORQUE := 0;
       #DIGITAL_INPUTS := 0;
   END_IF;
END_REGION
END_FUNCTION

ORGANIZATION_BLOCK "Main"   // OB1, FBD
TITLE = "Main Program Sweep (Cycle)"
{ S7_Optimized_Access := 'FALSE' }
VERSION : 0.1
// This sample program only demonstrates the basic approach. We do not accept any legal or other liability for incorrect program functions and their consequences!
   VAR_TEMP
      OB1_EV_CLASS : Byte;   // Bits 0-3 = 1 (Coming event), Bits 4-7 = 1 (Event class 1)
      OB1_SCAN_1 : Byte;   // 1 (Cold restart scan 1 of OB 1), 3 (Scan 2-n of OB 1)
      OB1_PRIORITY : Byte;   // Priority of OB Execution
      OB1_OB_NUMBR : Byte;   // 1 (Organization block 1, OB1)
      OB1_RESERVED_1 : Byte;   // Reserved for system
      OB1_RESERVED_2 : Byte;   // Reserved for system
      OB1_PREV_CYCLE : Int;   // Cycle time of previous OB1 scan (milliseconds)
      OB1_MIN_CYCLE : Int;   // Minimum cycle time of OB1 (milliseconds)
      OB1_MAX_CYCLE : Int;   // Maximum cycle time of OB1 (milliseconds)
      OB1_DATE_TIME : Date_And_Time;   // Date and time OB1 started
   END_VAR
BEGIN

REGION Network 1: Control of the drive velocity-UDT-S73xx
   // Please take note of the manual "MOVIKIT® Positioning, Velocity"
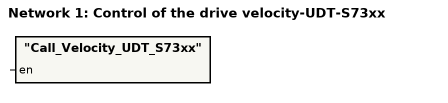
   "Call_Velocity_UDT_S73xx"();
END_REGION
END_ORGANIZATION_BLOCK